		IF (SIf.Cfg.bolEnableLampTest) THEN
			//--------------------------------------------------------------------------------------
			// sub state machine for lamp test sequence
			CASE me.SubStateMachine.intState OF
				cSTA_SUB_INITIALIZED:
					me.SubStateMachine.intStateNext := cSTA_SUB_TestGreen;
				cSTA_SUB_TestGreen:
					SIf.Out.bolGreen.intern := TRUE;
					IF (me.SubStateMachine.udiTimeInState_ms > SIf.Par.udiLampTestTime_ms) THEN 
						me.SubStateMachine.intStateNext := cSTA_SUB_TestYellow;
					END_IF
				cSTA_SUB_TestYellow:
					SIf.Out.bolYellow.intern := TRUE;
					IF (me.SubStateMachine.udiTimeInState_ms > SIf.Par.udiLampTestTime_ms) THEN 
						me.SubStateMachine.intStateNext := cSTA_SUB_TestRed;
					END_IF			
				cSTA_SUB_TestRed:
					SIf.Out.bolRed.intern := TRUE;
					IF (me.SubStateMachine.udiTimeInState_ms > SIf.Par.udiLampTestTime_ms) THEN 
						me.SubStateMachine.intStateNext := cSTA_SUB_TestBeep;
					END_IF				
				cSTA_SUB_TestBeep:
					SIf.Out.bolBeep.intern := TRUE;
					IF (me.SubStateMachine.udiTimeInState_ms > SIf.Par.udiLampTestTime_ms) THEN
						SIf.Out.bolGreen.intern := FALSE;
						SIf.Out.bolYellow.intern := FALSE;
						SIf.Out.bolRed.intern := FALSE;
						SIf.Out.bolBeep.intern := FALSE; 
						me.SubStateMachine.intStateNext := cSTA_SUB_FINISH;
					END_IF				
				cSTA_SUB_FINISH:
					;
				
			END_CASE
		ELSE // Lamp test not enabled, PONBusy is done
			me.SubStateMachine.intStateNext := cSTA_SUB_FINISH;
		END_IF

		
		// State Change Condition
		IF (me.SubStateMachine.intState = cSTA_SUB_FINISH) THEN	// Test done
			me.StateMachine.intStateNext :=  cSTA_PON;
		END_IF
	END_IF




//--------------------------------------------------------------------------------------
// Exit action
	IF (me.StateMachine.intState<>me.StateMachine.intStateNext) THEN
		;
	END_IF
END_METHOD

METHOD PROTECTED sta_RUN : BOOL
// state implemetation
//--------------------------------------------------------------------------------------
// Entry action
	IF (me.StateMachine.intState<>me.StateMachine.intStateLastCycle) THEN
		me.StateMachine.intStateLastCycle := me.StateMachine.intState;

	END_IF


//--------------------------------------------------------------------------------------
// Cyclic action
	IF (me.StateMachine.intState=me.StateMachine.intStateLastCycle) THEN

		// Simulation
		IF (CIf.SwCfg.bolSimulation) THEN
			;
		END_IF
		
		// Oscillator for blinking lamp
		IF (udiTimer >= 2*SIf.Par.udiBlinkTime_ms) THEN
			bolTimer:= FALSE;
			udiTimer:= 0;
		ELSIF (udiTimer >= SIf.Par.udiBlinkTime_ms) THEN
			bolTimer:= TRUE;
		END_IF
		udiTimer:= udiTimer + me.FUBInfo.udiSample_ms;
		// Oscillator for Beep
		IF (udiBeepTimer >= (SIf.Par.udiBeepOffTime_ms + SIf.Par.udiBeepOnTime_ms)) THEN
			bolBeepTimer:= TRUE;
			udiBeepTimer:= 0;
		ELSIF (udiBeepTimer >= SIf.Par.udiBeepOnTime_ms) THEN
			bolBeepTimer:= FALSE;
		END_IF
		udiBeepTimer:= udiBeepTimer + me.FUBInfo.udiSample_ms;	
		
		// Green Lamp
		SIf.Out.bolGreen.intern := setLampOutput(bolBlink:= In_bolGreenBlink, bolOn:= In_bolGreenOn, uinCnt:= In_uinCntGreen, 
												uinCntOLD:= uin_InCntGreenOld, bolOscillator:= bolTimer);
		// Yellow Lamp
		SIf.Out.bolYellow.intern := setLampOutput(bolBlink:= In_bolYellowBlink, bolOn:= In_bolYellowOn, uinCnt:= In_uinCntYellow, 
												uinCntOLD:= uin_InCntYellowOld, bolOscillator:= bolTimer);
		// Red Lamp
		SIf.Out.bolRed.intern := setLampOutput(bolBlink:= In_bolRedBlink, bolOn:= In_bolRedOn, uinCnt:= In_uinCntRed, 
												uinCntOLD:= uin_InCntRedOld, bolOscillator:= bolTimer);
		// Beep										
		SIf.Out.bolBeep.intern := setBeepOutput(bolOscillate:= In_bolBeepOn, uinCnt:= In_uinCntBeep,
												uinCntOLD:= uin_InCntBeepOld, bolOscillator:= bolBeepTimer);
												
		// Reset
		IF (CIf.Job.bolAlmReset) THEN
			uin_InCntGreenOld:= In_uinCntGreen;
			uin_InCntYellowOld:= In_uinCntYellow;
			uin_InCntRedOld:= In_uinCntRed;
			uin_InCntBeepOld:= In_uinCntBeep;
			CIf.Job.bolAlmReset := FALSE;
		END_IF
		
		// State Change Condition
		IF(me.intCmd=cCMD_OFF) THEN
			me.StateMachine.intStateNext := cSTA_OFFBusy;
		END_IF
	END_IF



//--------------------------------------------------------------------------------------
// Exit action
	IF (me.StateMachine.intState<>me.StateMachine.intStateNext) THEN
		;
	END_IF
END_METHOD

METHOD PROTECTED sta_RUNBusy : BOOL
// state implemetation
//--------------------------------------------------------------------------------------
// Entry action
	IF (me.StateMachine.intState<>me.StateMachine.intStateLastCycle) THEN
		me.StateMachine.intStateLastCycle := me.StateMachine.intState;

	END_IF


//--------------------------------------------------------------------------------------
// Cyclic action
	IF (me.StateMachine.intState=me.StateMachine.intStateLastCycle) THEN

		
		// State Change Condition
		IF (TRUE) THEN
			me.StateMachine.intStateNext := cSTA_RUN;
		END_IF
	END_IF


//--------------------------------------------------------------------------------------
// Exit action
	IF (me.StateMachine.intState<>me.StateMachine.intStateNext) THEN
		;
	END_IF
END_METHOD

METHOD PROTECTED StateMachine : BOOL
SUPER^.StateMachine();

// main statemachine of base controller
CASE me.StateMachine.intState OF
	cSTA_RUN:
		THIS^.sta_RUN();
	cSTA_RUNBusy:
		THIS^.sta_RUNBusy();
END_CASE;
END_METHOD

END_FUNCTION_BLOCK

// POUs/Controller/Lvl0/UMC [Universal Motor Controller]/FB_UMC
FUNCTION_BLOCK FB_UMC EXTENDS FB_CtrlBase
VAR_INPUT
	In_uinStatus				: UINT;
	In_intMotorActualSpeed		: INT;
	In_uinMotorSetSpeed			: UINT;
	In_strNetId					: AMSNETID;
	In_uintPort					: WORD;
	In_uinECATState				: UINT;
	In_bolEmoOk					: BOOL;
END_VAR
VAR_OUTPUT
	Out_uinControl      	: UINT;
	Out_uinSpeedSetpoint	: UINT;
END_VAR
VAR
	/// Specific interface struct for public access
	SIf					: T_Ctrl_SIf_UMC;
	In_unStatus			: U_UMC_Lenze_Status;
	Out_unControl		: U_UMC_Lenze_Control;
	arTurnDirection		: ARRAY[0..MAX_E_TURN_DIRECTION] OF BOOL;
	fbPulse				: TC2_STANDARD.TP;
END_VAR
VAR CONSTANT
	cLEFT				: BOOL := TRUE;
	cRIGHT				: BOOL := FALSE;

	cEtherCAT_OP_MODE		: UINT := 16#0008;
	cEtherCAT_MODE_MASK		: UINT := 16#000F;
END_VAR

(*__________________________________________________________________________________________________
¦	
¦	Vistaprint Schweiz GmbH
¦	CH - 8401 Winterthur
¦
¦	www.vistaprint.ch - info@vistaprint.ch
¦___________________________________________________________________________________________________

Function desription:
Lenze Motor implementation. 


History:
Version		Date			Author		Comment
---------------------------------------------------------------------------------------------------
0.00.1		09.07.2013		PC			Start history
0.00.2		04.02.2014		AVM/MRU		Simulation mode
										cCMD_LEFT / cCMD_RIGHT added in FB_init / getCmdState

___________________________________________________________________________________________________*)


IF (me.bolActivate) THEN // cyclic call enabled
	IF (CIf.Info.bolInitDone=FALSE) THEN // first cycle -> init
		CtrlInit();
		CIf.Info.bolInitDone := TRUE;
	ELSE
		CycleStartDuty();
	
		Always();
		
		StateMachine();
		
		CycleEndDuty();
	END_IF
END_IF;

METHOD PROTECTED Always : BOOL
SUPER^.Always();

// ----------------------------------------------------------------------------------
// Simulation
IF (CIf.SwCfg.bolSimulation) THEN
	// Simulate inputs (no physical inputs)
	SIf.In.bolEmoOk.intern := TRUE;
END_IF

// ----------------------------------------------------------------------------------
// Conditions Always
IF (me.StateMachine.intState<>cSTA_SINGLE_ANSWER) THEN
	IF (((me.Alarm.eActivAlmClass=E_AlmClass.OFF) OR (me.intCmd=cCMD_OFF))
			AND (me.StateMachine.intState<>cSTA_ERROR) AND (me.StateMachine.intState<>cSTA_ERRORQuit)
			AND (me.StateMachine.intState<>cSTA_EOFF) AND (me.StateMachine.intState<>cSTA_EOFFBusy)
			AND (me.StateMachine.intState<>cSTA_OFF) AND (me.StateMachine.intState<>cSTA_OFFBusy)
			AND (me.StateMachine.intState<>UMC_CmdState.cSTA_RESETMOTORERROR) 
			AND (me.StateMachine.intState<>UMC_CmdState.cSTA_SETOPERATIONMODE)) THEN
		me.StateMachine.intStateNext := cSTA_OFFBusy;	
	END_IF

	//-------------------------------------------------------------------------------
	// Monitoring of inputs from Safety PLC (no physical inputs)
	//-------------------------------------------------------------------------------
	// Emergency Off
	IF ((SIf.In.bolEmoOk.intern = FALSE) AND (me.StateMachine.intState <> cSTA_EOFF) 
		AND (me.StateMachine.intState <> BASE_PLC.cSTA_EOFFBusy)
		AND (me.StateMachine.intState <> BASE_PLC.cSTA_ERROR) 
		AND (me.StateMachine.intState <> BASE_PLC.cSTA_PON) 
		AND (me.StateMachine.intState <> BASE_PLC.cSTA_PONBusy) 
		AND (me.StateMachine.intState<>BASE_PLC.cSTA_INITIALIZED)
		AND (me.StateMachine.intState <> BASE_PLC.cSTA_ERRORQuit)) THEN
		me.StateMachine.intStateNext := cSTA_EOFFBusy;				
	END_IF	
END_IF
END_METHOD

METHOD PROTECTED cmd_MotorOff : BOOL
Out_unControl.Output 				:= 0;
Out_unControl.Data.SetDCBreak 		:= 1;
Out_unControl.Data.SetHalt        	:= 1;
Out_unControl.Data.SetQuickStop    	:= 1;
SIf.Out.uinSpeedSetpoint.intern 	:= 0;
END_METHOD

METHOD PROTECTED cmd_MotorOn : BOOL
VAR_INPUT
	bDirection		: BOOL;		// Direction of the drive; False = Right; True = Left
	uinSpeed		: UINT;					// Speed of the belt
END_VAR
Out_unControl.Output 				:= 0;
Out_unControl.Data.EnableOperation 	:= 1;
Out_unControl.Data.SwitchOn        	:= 1;
Out_unControl.Data.SetSpeedCcw     	:= bDirection;

SIf.Out.uinSpeedSetpoint.intern 	:= uinSpeed;
END_METHOD

METHOD PROTECTED cmd_MotorReset : BOOL
VAR_INPUT
END_VAR
cmd_MotorOff();
Out_unControl.Data.ResetFault 		:= 1;
END_METHOD

METHOD PROTECTED cmd_MotorStop : BOOL
VAR_INPUT
END_VAR
Out_unControl.Output 				:= 0;
Out_unControl.Data.SetDCBreak 		:= 1;
Out_unControl.Data.SetHalt        	:= 1;
Out_unControl.Data.SetQuickStop    	:= 1;
END_METHOD

METHOD PROTECTED CtrlInit : BOOL
VAR_INPUT
END_VAR
SUPER^.CtrlInit();

arTurnDirection[E_TURN_DIRECTION.AUTOMATIC] := FALSE;
arTurnDirection[E_TURN_DIRECTION.LEFT] 		:= FALSE;
arTurnDirection[E_TURN_DIRECTION.RIGHT] 	:= TRUE;

SIf.Cur.uinSpeedLimit := SIf.Cfg.uinMaxSpeed * SIf.Cfg.uinLC11_100 / 100;
END_METHOD

PROPERTY PUBLIC CtrlSIf : POINTER TO T_Ctrl_SIf_UMC
GET
CtrlSIf := ADR(SIf);
END_GET
SET
END_SET
END_PROPERTY

METHOD PROTECTED CycleEndDuty : BOOL
VAR_INPUT
END_VAR
SIf.Out.uinControl.intern := Out_unControl.Output;

SUPER^.CycleEndDuty();
END_METHOD

METHOD PROTECTED CycleStartDuty : BOOL
VAR_INPUT
END_VAR
SUPER^.CycleStartDuty();

In_unStatus.Input := SIf.In.uinStatus.intern;
END_METHOD

METHOD FB_init : BOOL
VAR_INPUT
	bInitRetains : BOOL; // if TRUE, the retain variables are initialized (warm start / cold start)
	bInCopyCode : BOOL;  // if TRUE, the instance afterwards gets moved into the copy code (online change)
END_VAR
VAR
	iIdx		: UINT;
	iLength		: UINT;	
END_VAR
//------------------------------------------------------------------------------------------------------------------------
// to manually change in new FUB implementation!!!
// define valid commands for this controller
iLength := SIZEOF(CIf.Job.aCmdList)/SIZEOF(CIf.Job.aCmdList[0]);
iIdx := 0;

WHILE (iIdx < iLength) AND (CIf.Job.aCmdList[iIdx].intCmd <> cCMD_INITIALIZED) DO
	iIdx := iIdx + 1; 
END_WHILE

IF (iIdx < iLength) THEN
// Add configuration of own comands	
	CIf.Job.aCmdList[iIdx].intCmd := BASE_PLC.cCMD_STOP;
	CIf.Job.aCmdList[iIdx].strName := 'Stop'; 
	CIf.Job.aCmdList[iIdx].bolAvailable := TRUE;
	iIdx := iIdx + 1;
	CIf.Job.aCmdList[iIdx].intCmd := cCMD_RUN;
	CIf.Job.aCmdList[iIdx].strName := 'Run'; 
	CIf.Job.aCmdList[iIdx].bolAvailable := TRUE;
	iIdx := iIdx + 1;
	CIf.Job.aCmdList[iIdx].intCmd := cCMD_LEFT;
	CIf.Job.aCmdList[iIdx].strName := 'Left'; 
	CIf.Job.aCmdList[iIdx].bolAvailable := TRUE;
	iIdx := iIdx + 1;
	CIf.Job.aCmdList[iIdx].intCmd := cCMD_RIGHT;
	CIf.Job.aCmdList[iIdx].strName := 'Right'; 
	CIf.Job.aCmdList[iIdx].bolAvailable := TRUE;
	iIdx := iIdx + 1;
ELSE
	;// Error if the aCmdList Array is to small
END_IF

// set name of class/typ
CIf.Info.strType := 'FB_UMC'; 

// set alarm class
SIf.Alm[E_ALM_UMC.MotorOnTimeout].eAlmClass := Base_PLC.E_AlmClass.TSTOP;
SIf.Alm[E_ALM_UMC.MotorOnTimeout].strText := 'Motor On Timeout'; 
SIf.Alm[E_ALM_UMC.MotorError].eAlmClass := Base_PLC.E_AlmClass.TSTOP;
SIf.Alm[E_ALM_UMC.MotorError].strText := 'Motor Error';
SIf.Alm[E_ALM_UMC.MotorWarning].eAlmClass := Base_PLC.E_AlmClass.WARNING;
SIf.Alm[E_ALM_UMC.MotorWarning].strText := 'Motor Warning';
SIf.Alm[E_ALM_UMC.MotorOverCurrent].eAlmClass := Base_PLC.E_AlmClass.WARNING;
SIf.Alm[E_ALM_UMC.MotorOverCurrent].strText := 'Motor Over Current';
SIf.Alm[E_ALM_UMC.MotorNotReady].eAlmClass := Base_PLC.E_AlmClass.TSTOP;
SIf.Alm[E_ALM_UMC.MotorNotReady].strText := 'Motor Not Ready';
SIf.Alm[E_ALM_UMC.DirectionParameterOverflow].eAlmClass := Base_PLC.E_AlmClass.TSTOP;
SIf.Alm[E_ALM_UMC.DirectionParameterOverflow].strText := 'Direction Parameter Overflow';
SIf.Alm[E_ALM_UMC.SpeedOverLimit].eAlmClass := Base_PLC.E_AlmClass.WARNING;
SIf.Alm[E_ALM_UMC.SpeedOverLimit].strText := 'Motor Setpoint over the limit';

//*******************************************************************************
// initial values
//*******************************************************************************

// software configuration
CIf.SwCfg.bolExist := TRUE;
CIf.SwCfg.bolEnable := TRUE;
CIf.SwCfg.bolSimulation := FALSE;

// configuration
SIf.Cfg.uinLC11 := 1500;
SIf.Cfg.uinLC11_100 := 16384;
SIf.Cfg.uinMaxSpeed := 150;

// parameter
SIf.Par.udiStartupOnTime_ms := 5000;
SIf.Par.udiMotorOnTime_ms 	:= 10000;
SIf.Par.uinSpeed_rpm 		:= 1000;
SIf.Par.uinMotorResetPulseTime_ms	:= 500;
SIf.Par.uinMotorResetCnt 		:= 3;
SIf.Par.udiMoveStartLatency 	:= 15;
SIf.Par.udiMoveStopLatency 		:= 60;
SIf.Par.eRotationDirection  := E_TURN_DIRECTION.LEFT;

SIf.Par.udiSimMotorOnTime_ms := SIf.Par.udiMotorOnTime_ms / 10;
END_METHOD

METHOD PROTECTED getCmdState : STRING

VAR_INPUT
	intCmdState: INT;
	bolState: BOOL;
END_VAR
getCmdState := SUPER^.getCmdState(intCmdState:=intCmdState,bolState:=bolState); // get global/base defined cmds/states

IF (getCmdState='') THEN // global not defined get local
	// get string cmd/state string information in runtime
	IF (bolState=FALSE) THEN
		// Comands's
		CASE intCmdState OF
			cCMD_LEFT: 
				getCmdState := 'cCMD_Left';
			cCMD_RIGHT: 
				getCmdState := 'cCMD_Right';
		END_CASE;
	ELSE
		// States's
		CASE intCmdState OF
			cSTA_RUN: 
				getCmdState := 'RUN';
			cSTA_RUNBusy: 
				getCmdState := 'RUNBusy';
			UMC_CmdState.cSTA_RESETMOTORERROR:
				getCmdState := 'RESETMOTORERROR';
			UMC_CmdState.cSTA_SETOPERATIONMODE:
				getCmdState := 'SETOPERATIONMODE';
		END_CASE;
	END_IF
END_IF
END_METHOD

METHOD getCtrlSIf : POINTER TO T_Ctrl_SIf_UMC
getCtrlSIf := ADR(SIf);
END_METHOD

METHOD PROTECTED GetMotorStatus : E_UMC_MOTOR_STATUS
VAR_INPUT
	uinMotorStatus		: UINT;
END_VAR
uinMotorStatus := uinMotorStatus AND 16#0F00;
uinMotorStatus := SHR(uinMotorStatus,8);
GetMotorStatus := UINT_TO_INT(uinMotorStatus);
END_METHOD

METHOD PROTECTED GetSpeedValue : UINT
VAR
	uinSpeedOutput			: UINT;
END_VAR
uinSpeedOutput := SIf.Par.uinSpeed_rpm * SIf.Cfg.uinLC11_100 / SIf.Cfg.uinLC11;

IF uinSpeedOutput > SIf.Cur.uinSpeedLimit THEN
	uinSpeedOutput := SIf.Cur.uinSpeedLimit;
	pfbAlarmCtrl^.setAlarm(CIf.Info.intCtrlId,INT_TO_UINT(E_ALM_UMC.SpeedOverLimit),0,ADR(SIf.Alm),E_AlmState.RST,CIf.Job.eMe_ActivAlmClass);
END_IF

GetSpeedValue := uinSpeedOutput;
END_METHOD

METHOD PROTECTED IoInBridge : BOOL
// digitale and analoge inputs read from hardware or forcing
SIf.In.uinStatus.map			:= THIS^.In_uinStatus				;
SIf.In.intMotorActualSpeed.map	:= THIS^.In_intMotorActualSpeed	;
SIf.In.uinMotorSetSpeed.map		:= THIS^.In_uinMotorSetSpeed		;
SIf.In.bolEmoOk.map				:= THIS^.In_bolEmoOk		;

IF (CIf.SwCfg.bolSimulation = FALSE) THEN
	BASE_PLC.getInUint(CIf.Job.bolIoForce,ADR(SIf.In.uinStatus));
	BASE_PLC.getInUint(CIf.Job.bolIoForce,ADR(SIf.In.intMotorActualSpeed));
	BASE_PLC.getInUint(CIf.Job.bolIoForce,ADR(SIf.In.uinMotorSetSpeed));
	BASE_PLC.getInUint(CIf.Job.bolIoForce,ADR(SIf.In.bolEmoOk));
ELSE
	//simulation of global IO
END_IF
END_METHOD

METHOD PROTECTED IoOutBridge : BOOL
VAR
	bolSwitchValvesOff: BOOL;
END_VAR
// digitale and analoge inputs read from hardware or forcing
IF (CIf.SwCfg.bolSimulation = FALSE) THEN
	BASE_PLC.setOutUint(CIf.Job.bolIoForce ,ADR(SIf.Out.uinControl));
	BASE_PLC.setOutUint(CIf.Job.bolIoForce ,ADR(SIf.Out.uinSpeedSetpoint));

	THIS^.Out_uinControl			:= SIf.Out.uinControl.map	;
	THIS^.Out_uinSpeedSetpoint		:= SIf.Out.uinSpeedSetpoint.map	;
END_IF
END_METHOD

METHOD PROTECTED sta_EOFF : BOOL
VAR_INPUT
END_VAR
// state implemetation
//--------------------------------------------------------------------------------------
// Entry action
	IF (me.StateMachine.intState<>me.StateMachine.intStateLastCycle) THEN
		me.StateMachine.intStateLastCycle := me.StateMachine.intState;	
	END_IF

//--------------------------------------------------------------------------------------
// Cyclic action
	IF (me.StateMachine.intState=me.StateMachine.intStateLastCycle) THEN		
		// As long as the EMO is not reseted!
		IF SIf.In.bolEmoOk.intern THEN
			me.StateMachine.intStateNext := BASE_PLC.cSTA_OFFBusy;			
		ELSE
			IF me.intCmd <> BASE_PLC.cCMD_OFF THEN
				// Clear pending and new commands cyclic to prevent automatic recovery!	
				CIf.Job.intACmd := BASE_PLC.cCMD_DONE;
				CIf.Job.intMCmd := BASE_PLC.cCMD_DONE;		
			END_IF
		END_IF
	END_IF

//--------------------------------------------------------------------------------------
// Exit action
	IF (me.StateMachine.intState<>me.StateMachine.intStateNext) THEN
		;
	END_IF
END_METHOD

METHOD PROTECTED sta_EOFFbusy : BOOL
VAR_INPUT
END_VAR
// state implemetation
//--------------------------------------------------------------------------------------
// Entry action
IF (me.StateMachine.intState<>me.StateMachine.intStateLastCycle) THEN
	me.StateMachine.intStateLastCycle := me.StateMachine.intState;
	cmd_MotorOff();
END_IF

//--------------------------------------------------------------------------------------
// Cyclic action
IF (me.StateMachine.intState=me.StateMachine.intStateLastCycle) THEN
	IF (TRUE) THEN
		me.StateMachine.intStateNext := BASE_PLC.cSTA_EOFF;
	END_IF
END_IF

//--------------------------------------------------------------------------------------
// Exit action
IF (me.StateMachine.intState<>me.StateMachine.intStateNext) THEN
	;
END_IF
END_METHOD

METHOD PROTECTED sta_ERROR : BOOL
// state implemetation
//--------------------------------------------------------------------------------------
// Entry action
	IF (me.StateMachine.intState<>me.StateMachine.intStateLastCycle) THEN
		me.StateMachine.intStateHistory := me.StateMachine.intStateLastCycle; // -> possibillity to go back to state before error
		me.StateMachine.intStateLastCycle := me.StateMachine.intState;
		SIf.Cur.uinMotorResetCnt := 0;
		cmd_MotorOff();
	END_IF


//--------------------------------------------------------------------------------------
// Cyclic action
	IF (me.StateMachine.intState=me.StateMachine.intStateLastCycle) THEN
		
		;
		
		
		// State Change Condition
		IF (CIf.Job.bolAlmReset = TRUE) THEN
			me.StateMachine.intStateNext := cSTA_ERRORQuit;
		END_IF
	END_IF




//--------------------------------------------------------------------------------------
// Exit action
	IF (me.StateMachine.intState<>me.StateMachine.intStateNext) THEN
		;
	END_IF
END_METHOD

METHOD PROTECTED sta_ERRORQuit : BOOL
// state implemetation
//--------------------------------------------------------------------------------------
// Entry action
	IF (me.StateMachine.intState<>me.StateMachine.intStateLastCycle) THEN
		me.StateMachine.intStateLastCycle := me.StateMachine.intState;
		
	END_IF


//--------------------------------------------------------------------------------------
// Cyclic action
	IF (me.StateMachine.intState=me.StateMachine.intStateLastCycle) THEN
		
		;
		// evtl. wait time if reset of device is necessary and then decide to go to states or ERROR state
		IF (CIf.Job.bolAlmReset = TRUE) THEN
			CIf.Job.eMe_ActivAlmClass := E_AlmClass.NONE; // reset feedback channel for parent
			CIf.Job.bolAlmReset := FALSE;
		END_IF
		
		// State Change Condition
		IF (CIf.Job.bolAlmReset = FALSE) THEN
			IF (me.StateMachine.intStateHistory<=cSTA_PON) THEN
				me.StateMachine.intStateNext := cSTA_PON;
			ELSIF (CIf.SwCfg.bolSimulation = TRUE) THEN	// Do not set operation mode in simulation
				me.StateMachine.intStateNext := BASE_PLC.cSTA_OFF;
			ELSE
				me.StateMachine.intStateNext := UMC_CmdState.cSTA_SETOPERATIONMODE;
			END_IF
		END_IF
	END_IF




//--------------------------------------------------------------------------------------
// Exit action
	IF (me.StateMachine.intState<>me.StateMachine.intStateNext) THEN
		;
	END_IF
END_METHOD

METHOD PROTECTED sta_OFF : BOOL
VAR_INPUT
END_VAR
// state implemetation
//--------------------------------------------------------------------------------------
// Entry action
	IF (me.StateMachine.intState<>me.StateMachine.intStateLastCycle) THEN
		me.StateMachine.intStateLastCycle := me.StateMachine.intState;

		SIf.Cur.uinMotorResetCnt := 0;
	END_IF


//--------------------------------------------------------------------------------------
// Cyclic action
	IF (me.StateMachine.intState=me.StateMachine.intStateLastCycle) THEN
		CASE me.intCmd OF
			cCMD_Left:
				SIf.Par.eRotationDirection := E_TURN_DIRECTION.LEFT;
				me.StateMachine.intStateNext := cSTA_RUNBusy;
			cCMD_Right:
				SIf.Par.eRotationDirection := E_TURN_DIRECTION.RIGHT;
				me.StateMachine.intStateNext := cSTA_RUNBusy;
			BASE_PLC.cCMD_STOP:
				me.StateMachine.intStateNext := BASE_PLC.cSTA_STOPBusy;
			BASE_PLC.cCMD_RUN:
				me.StateMachine.intStateNext := cSTA_RUNBusy;
		END_CASE
	END_IF


//--------------------------------------------------------------------------------------
// Exit action
	IF (me.StateMachine.intState<>me.StateMachine.intStateNext) THEN
		;
	END_IF
END_METHOD

METHOD PROTECTED sta_OFFBusy : BOOL
VAR
	uinECatStatus	: UINT;
	eMotorStatus	: E_UMC_MOTOR_STATUS;
END_VAR
// state implemetation
//--------------------------------------------------------------------------------------
// Entry action
	IF (me.StateMachine.intState<>me.StateMachine.intStateLastCycle) THEN
		me.StateMachine.intStateLastCycle := me.StateMachine.intState;
		cmd_MotorOff();
	END_IF


//--------------------------------------------------------------------------------------
// Cyclic action
	IF (me.StateMachine.intState=me.StateMachine.intStateLastCycle) THEN
		eMotorStatus := GetMotorStatus(sif.In.uinStatus.intern);
		uinECatStatus := In_uinECATState AND cEtherCAT_MODE_MASK;

		IF    (uinECatStatus = cEtherCAT_OP_MODE)
		  AND NOT In_unStatus.Data.Trouble 
		  AND In_unStatus.Data.ActSpeedIsZero
		  AND (eMotorStatus = E_UMC_MOTOR_STATUS.ReadyToSwitchON) THEN
			me.StateMachine.intStateNext := Base_PLC.cSTA_OFF;
		ELSIF (CIf.SwCfg.bolSimulation = TRUE) THEN	// Do not set operation mode in simulation
			me.StateMachine.intStateNext := BASE_PLC.cSTA_OFF;
		ELSE
			IF me.StateMachine.udiTimeInState_ms > SIf.Par.uinMotorResetPulseTime_ms THEN
				IF SIf.Cur.uinMotorResetCnt > SIf.Par.uinMotorResetCnt THEN
					pfbAlarmCtrl^.setAlarm(CIf.Info.intCtrlId,INT_TO_UINT(E_ALM_UMC.MotorError),0,ADR(SIf.Alm),E_AlmState.RST,CIf.Job.eMe_ActivAlmClass);
					me.StateMachine.intStateNext := Base_PLC.cSTA_ERROR;	
				ELSE
					me.StateMachine.intStateNext := UMC_CmdState.cSTA_SETOPERATIONMODE;
				END_IF
			END_IF
		END_IF
	END_IF

//--------------------------------------------------------------------------------------
// Exit action
	IF (me.StateMachine.intState<>me.StateMachine.intStateNext) THEN
		;
	END_IF
END_METHOD

METHOD PROTECTED sta_PON : BOOL
VAR_INPUT
END_VAR
// state implemetation
//--------------------------------------------------------------------------------------
// Entry action
	IF (me.StateMachine.intState<>me.StateMachine.intStateLastCycle) THEN
		me.StateMachine.intStateLastCycle := me.StateMachine.intState;
		
	END_IF


//--------------------------------------------------------------------------------------
// Cyclic action
	IF (me.StateMachine.intState=me.StateMachine.intStateLastCycle) THEN
		;
	END_IF




//--------------------------------------------------------------------------------------
// Exit action
	IF (me.StateMachine.intState<>me.StateMachine.intStateNext) THEN
		;
	END_IF
END_METHOD

METHOD PROTECTED sta_RESETMOTORERROR : BOOL
VAR
	eMotorStatus	: E_UMC_MOTOR_STATUS;
END_VAR
// state implemetation
//--------------------------------------------------------------------------------------
// Entry action
	IF (me.StateMachine.intState<>me.StateMachine.intStateLastCycle) THEN
		me.StateMachine.intStateLastCycle := me.StateMachine.intState;
		cmd_MotorReset();
	END_IF


//--------------------------------------------------------------------------------------
// Cyclic action
	IF (me.StateMachine.intState=me.StateMachine.intStateLastCycle) THEN
		eMotorStatus := GetMotorStatus(sif.In.uinStatus.intern);

		IF me.SubStateMachine.udiTimeInState_ms > SIf.Par.uinMotorResetPulseTime_ms THEN
			SIf.Cur.uinMotorResetCnt := SIf.Cur.uinMotorResetCnt + 1;
			me.StateMachine.intStateNext := BASE_PLC.cSTA_OFFBusy;
		END_IF
	END_IF


//--------------------------------------------------------------------------------------
// Exit action
	IF (me.StateMachine.intState<>me.StateMachine.intStateNext) THEN
		Out_unControl.Data.ResetFault := FALSE;
	END_IF
END_METHOD

METHOD PROTECTED sta_RUN : BOOL
VAR
	uniStatus 		: U_UMC_Lenze_Status;
END_VAR
// state implemetation
//--------------------------------------------------------------------------------------
// Entry action
	IF (me.StateMachine.intState<>me.StateMachine.intStateLastCycle) THEN
		me.StateMachine.intStateLastCycle := me.StateMachine.intState;
		CIf.Job.intACmd := BASE_PLC.cCMD_DONE;
	END_IF


//--------------------------------------------------------------------------------------
// Cyclic action
	IF (me.StateMachine.intState=me.StateMachine.intStateLastCycle) THEN
		IF In_unStatus.Data.Trouble THEN
			pfbAlarmCtrl^.setAlarm(CIf.Info.intCtrlId,INT_TO_UINT(E_ALM_UMC.MotorError),0,ADR(SIf.Alm),E_AlmState.RST,CIf.Job.eMe_ActivAlmClass);
			me.StateMachine.intStateNext := Base_PLC.cSTA_ERROR;	
		END_IF
		
		IF (me.StateMachine.intStateNext <> Base_PLC.cSTA_ERROR) THEN
			// Reenter the RunBusy state again if the speed changes
			IF SIf.Par.uinSpeed_rpm <> SIf.Cur.uinSpeed_rpm THEN
				me.StateMachine.intStateNext := cSTA_RUNBusy;
			END_IF
			
			// Reenter the RunBusy state again if the direction changes.
			IF SIf.Par.eRotationDirection <> SIf.Cur.eDirection THEN
				me.StateMachine.intStateNext := cSTA_RUNBusy;
			END_IF

			CASE me.intCmd OF
				cCMD_Left:
					SIf.Par.eRotationDirection := E_TURN_DIRECTION.LEFT;
					me.StateMachine.intStateNext := cSTA_RUNBusy;
				cCMD_Right:
					SIf.Par.eRotationDirection := E_TURN_DIRECTION.RIGHT;
					me.StateMachine.intStateNext := cSTA_RUNBusy;
				BASE_PLC.cCMD_STOP:
					me.StateMachine.intStateNext := BASE_PLC.cSTA_STOPBusy;
			END_CASE
		END_IF
END_IF


//--------------------------------------------------------------------------------------
// Exit action
	IF (me.StateMachine.intState<>me.StateMachine.intStateNext) THEN
		;
	END_IF
END_METHOD

METHOD PROTECTED sta_RUNBusy : BOOL
VAR
	uniStatus 		: U_UMC_Lenze_Status;
END_VAR
// state implemetation
//--------------------------------------------------------------------------------------
// Entry action
	IF (me.StateMachine.intState<>me.StateMachine.intStateLastCycle) THEN
		me.StateMachine.intStateLastCycle := me.StateMachine.intState;

		SIf.Cur.uinSpeed_rpm := SIf.Par.uinSpeed_rpm;
		SIf.Cur.uinSpeedOuput := GetSpeedValue();
		SIf.Cur.eDirection 	:= SIf.Par.eRotationDirection;
		
		// Switch Motor ON
		IF SIf.Par.eRotationDirection < E_TURN_DIRECTION.MAX_E_TURN_DIRECTION THEN
			cmd_MotorOn(arTurnDirection[SIf.Par.eRotationDirection], SIf.Cur.uinSpeedOuput);
		ELSE
			pfbAlarmCtrl^.setAlarm(CIf.Info.intCtrlId,INT_TO_UINT(E_ALM_UMC.DirectionParameterOverflow),0,ADR(SIf.Alm),E_AlmState.RST,CIf.Job.eMe_ActivAlmClass);
			me.StateMachine.intStateNext := Base_PLC.cSTA_ERROR;	
		END_IF

		fbSimulationTimer.IN := FALSE;
		fbSimulationTimer.PT := UDINT_TO_TIME(SIf.Par.udiSimMotorOnTime_ms);
		fbSimulationTimer(); // set time/reset timer
		fbSimulationTimer.IN := TRUE; // start timer

	END_IF


//--------------------------------------------------------------------------------------
// Cyclic action
	IF (me.StateMachine.intState=me.StateMachine.intStateLastCycle) THEN
		IF (CIf.SwCfg.bolSimulation) THEN
			fbSimulationTimer(); // simulation time
			IF (fbSimulationTimer.Q) THEN
				SIf.In.uinMotorSetSpeed.intern 	:= SIf.Out.uinSpeedSetpoint.intern;
				SIf.In.uinMotorSetSpeed.intern 	:= SIf.Out.uinSpeedSetpoint.intern;
				uniStatus.Input 				:= 0;
				uniStatus.Data.DriveReady		:= 1;
				uniStatus.Data.SpeedActEqualSet := 1;
				uniStatus.Data.SpeedSetReached  := 1;
				uniStatus.Data.Status_1			:= 1;
				uniStatus.Data.Status_3			:= 1;
				uniStatus.Data.SpeedCcw			:= arTurnDirection[SIf.Par.eRotationDirection];
				SIf.In.uinStatus.intern 		:= uniStatus.Input;
			END_IF
		END_IF

		IF (me.StateMachine.udiTimeInState_ms > SIf.Par.udiMotorOnTime_ms) THEN
			pfbAlarmCtrl^.setAlarm(CIf.Info.intCtrlId,INT_TO_UINT(E_ALM_UMC.MotorOnTimeout),0,ADR(SIf.Alm),E_AlmState.RST,CIf.Job.eMe_ActivAlmClass);
			me.StateMachine.intStateNext := Base_PLC.cSTA_ERROR;	
		END_IF

		IF In_unStatus.Data.Trouble THEN
			pfbAlarmCtrl^.setAlarm(CIf.Info.intCtrlId,INT_TO_UINT(E_ALM_UMC.MotorError),0,ADR(SIf.Alm),E_AlmState.RST,CIf.Job.eMe_ActivAlmClass);
			me.StateMachine.intStateNext := Base_PLC.cSTA_ERROR;	
		END_IF
		
		IF (me.StateMachine.intStateNext <> Base_PLC.cSTA_ERROR) THEN
			IF (NOT In_unStatus.Data.Trouble) 
				AND (THIS^.arTurnDirection[SIf.Cur.eDirection] = In_unStatus.Data.SpeedCcw)	THEN
//				AND (In_unStatus.Data.SpeedSetReached) THEN
				me.StateMachine.intStateNext := cSTA_RUN;
			END_IF;	

			// Reenter the RunBusy state again if the speed changes
			IF GetSpeedValue() <> SIf.Cur.uinSpeedOuput THEN
				me.StateMachine.intStateLastCycle := -1;
			END_IF
			
			// Reenter the RunBusy state again if the direction changes.
			IF SIf.Par.eRotationDirection <> SIf.Cur.eDirection THEN
				me.StateMachine.intStateLastCycle := -1;
			END_IF
			
			CASE me.intCmd OF
				cCMD_Left:
					IF SIf.Par.eRotationDirection <> E_TURN_DIRECTION.LEFT THEN
						SIf.Par.eRotationDirection := E_TURN_DIRECTION.LEFT;
						me.StateMachine.intStateLastCycle := -1;
					END_IF
				cCMD_Right:
					IF SIf.Par.eRotationDirection <> E_TURN_DIRECTION.RIGHT THEN
						SIf.Par.eRotationDirection := E_TURN_DIRECTION.RIGHT;
						me.StateMachine.intStateLastCycle := -1;
					END_IF
				BASE_PLC.cCMD_STOP:
					me.StateMachine.intStateNext := BASE_PLC.cSTA_STOPBusy;
			END_CASE
		END_IF
END_IF


//--------------------------------------------------------------------------------------
// Exit action
	IF (me.StateMachine.intState<>me.StateMachine.intStateNext) THEN
		;
	END_IF
END_METHOD

METHOD PROTECTED sta_SETOPERATIONMODE : BOOL
VAR
	uinECatStatus		: UINT;

	fbEcReqSlaveState 	: FB_EcReqSlaveState;
	bExecute        	: BOOL;
	uinReqState     	: WORD := EC_DEVICE_STATE_OP;
	bError          	: BOOL;
	nErrId          	: UDINT;
END_VAR
// state implemetation
//--------------------------------------------------------------------------------------
// Entry action
	IF (me.StateMachine.intState<>me.StateMachine.intStateLastCycle) THEN
		me.StateMachine.intStateLastCycle := me.StateMachine.intState;
	END_IF


//--------------------------------------------------------------------------------------
// Cyclic action
	IF (me.StateMachine.intState=me.StateMachine.intStateLastCycle) THEN
		bExecute := NOT ((In_uinECATState AND cEtherCAT_MODE_MASK) = cEtherCAT_OP_MODE);

		IF NOT bExecute THEN
			me.StateMachine.intStateNext := UMC_CmdState.cSTA_RESETMOTORERROR;
		END_IF

		fbEcReqSlaveState(
			sNetId		:= F_CreateAmsNetId(In_strNetId), 
			nSlaveAddr	:= In_uintPort, 
			bExecute	:= bExecute, 
			state		:= uinReqState  );

		IF (me.StateMachine.udiTimeInState_ms > SIf.Par.udiStartupOnTime_ms) THEN
			pfbAlarmCtrl^.setAlarm(CIf.Info.intCtrlId,INT_TO_UINT(E_ALM_UMC.MotorError),0,ADR(SIf.Alm),E_AlmState.RST,CIf.Job.eMe_ActivAlmClass);
			me.StateMachine.intStateNext := Base_PLC.cSTA_ERROR;	
		END_IF
END_IF


//--------------------------------------------------------------------------------------
// Exit action
	IF (me.StateMachine.intState<>me.StateMachine.intStateNext) THEN
		Out_unControl.Data.ResetFault := FALSE;
	END_IF
END_METHOD

METHOD PROTECTED sta_STOP : BOOL
VAR_INPUT
END_VAR
// state implemetation
//--------------------------------------------------------------------------------------
// Entry action
	IF (me.StateMachine.intState<>me.StateMachine.intStateLastCycle) THEN
		me.StateMachine.intStateLastCycle := me.StateMachine.intState;

	END_IF


//--------------------------------------------------------------------------------------
// Cyclic action
	IF (me.StateMachine.intState=me.StateMachine.intStateLastCycle) THEN
		CASE me.intCmd OF
			cCMD_Left:
				SIf.Par.eRotationDirection := E_TURN_DIRECTION.LEFT;
				me.StateMachine.intStateNext := cSTA_RUNBusy;
			cCMD_Right:
				SIf.Par.eRotationDirection := E_TURN_DIRECTION.RIGHT;
				me.StateMachine.intStateNext := cSTA_RUNBusy;
			BASE_PLC.cCMD_RUN:
				me.StateMachine.intStateNext := cSTA_RUNBusy;
		END_CASE
	END_IF


//--------------------------------------------------------------------------------------
// Exit action
	IF (me.StateMachine.intState<>me.StateMachine.intStateNext) THEN
		;
	END_IF
END_METHOD

METHOD PROTECTED sta_STOPBusy : BOOL
VAR
	uniStatus 		: U_UMC_Lenze_Status;
END_VAR
// state implemetation
//--------------------------------------------------------------------------------------
// Entry action
	IF (me.StateMachine.intState<>me.StateMachine.intStateLastCycle) THEN
		me.StateMachine.intStateLastCycle := me.StateMachine.intState;
		// Switch Motor Off
		cmd_MotorStop();
	END_IF


//--------------------------------------------------------------------------------------
// Cyclic action
	IF (me.StateMachine.intState=me.StateMachine.intStateLastCycle) THEN
		IF (CIf.SwCfg.bolSimulation) THEN
			SIf.In.uinMotorSetSpeed.intern 	:= 0;
			SIf.In.intMotorActualSpeed.intern 	:= 0;
			uniStatus.Input 				:= 0;
			uniStatus.Data.ActSpeedIsZero	:= TRUE;
			SIf.In.uinStatus.intern 		:= uniStatus.Input;
		END_IF

		IF (me.StateMachine.udiTimeInState_ms < SIf.Par.udiMotorOnTime_ms) THEN
			IF (NOT In_unStatus.Data.Trouble) AND (In_unStatus.Data.ActSpeedIsZero) THEN
				me.StateMachine.intStateNext := Base_PLC.cSTA_STOP;
			END_IF;	
		ELSE
			pfbAlarmCtrl^.setAlarm(CIf.Info.intCtrlId,INT_TO_UINT(E_ALM_UMC.MotorError),0,ADR(SIf.Alm),E_AlmState.RST,CIf.Job.eMe_ActivAlmClass);
			me.StateMachine.intStateNext := Base_PLC.cSTA_ERROR;	
		END_IF
END_IF


//--------------------------------------------------------------------------------------
// Exit action
	IF (me.StateMachine.intState<>me.StateMachine.intStateNext) THEN
		Out_unControl.Data.ResetFault := FALSE;
	END_IF
END_METHOD

METHOD PROTECTED StateMachine : BOOL
SUPER^.StateMachine();

// main statemachine of base controller
CASE me.StateMachine.intState OF
	cSTA_RUNBusy:
		THIS^.sta_RUNBusy();
	cSTA_RUN:
		THIS^.sta_RUN();
	cSTA_STOPBusy: 
        THIS^.sta_STOPBusy();
    cSTA_STOP: 
        THIS^.sta_STOP();
	UMC_CmdState.cSTA_RESETMOTORERROR:
		THIS^.sta_RESETMOTORERROR();
	UMC_CmdState.cSTA_SETOPERATIONMODE:
		THIS^.sta_SETOPERATIONMODE();
END_CASE;
END_METHOD

END_FUNCTION_BLOCK

// POUs/Controller/Lvl0/VLV (Valve controller)/FB_VLV
FUNCTION_BLOCK FB_VLV EXTENDS FB_CtrlBase
VAR_INPUT
	In_bolOpened: BOOL;
	In_bolClosed: BOOL;
END_VAR
VAR_OUTPUT
	Out_bolOpen: BOOL;
	Out_bolClose: BOOL;
END_VAR
VAR
	/// Specific interface struct for public access
	SIf: T_Ctrl_SIf_VLV;
END_VAR

(*__________________________________________________________________________________________________
¦	
¦	Vistaprint Schweiz GmbH
¦	CH - 8401 Winterthur
¦
¦	www.vistaprint.ch - info@vistaprint.ch
¦___________________________________________________________________________________________________

Function desription:
Basic valve controller

History:
Version		Date			Author		Comment
---------------------------------------------------------------------------------------------------
0.00.1		06.03.2014		AVME/DSC	Start history. Based on CYL controller

___________________________________________________________________________________________________*)


IF (me.bolActivate) THEN // cyclic call enabled
	IF (CIf.Info.bolInitDone=FALSE) THEN // first cycle -> init
		CtrlInit();
		CIf.Info.bolInitDone := TRUE;
	ELSE
		CycleStartDuty();
	
		Always();
		
		StateMachine();
		
		CycleEndDuty();
	END_IF
END_IF;

METHOD PROTECTED Always : BOOL
IF (me.bolChangeBackToAUTO=TRUE) THEN // switch mode to automatic switch off controller
	//me.StateMachine.intStateNext := cSTA_OFFBusy;
	me.bolChangeBackToAUTO := FALSE; // for valve no change to off when switch to automatic!!
END_IF

SUPER^.Always();

// ----------------------------------------------------------------------------------
// cyclic actions outside of statemachine
IF (me.StateMachine.intState<>cSTA_SINGLE_ANSWER) THEN
	
	; // always error supervision
	// ----------------------------------------------------------------------------------
	// overrule error always from base -> no EOFF State!! in EOFF go to OFF
	IF (me.StateMachine.intStateNext = cSTA_EOFFBusy) THEN
		IF (me.StateMachine.intState=cSTA_OFF) THEN
			me.StateMachine.intStateNext := cSTA_OFF;
		ELSE // stay in OFF
			me.StateMachine.intStateNext := cSTA_OFFBusy;
		END_IF
	END_IF
END_IF
END_METHOD

METHOD FB_init : BOOL
VAR_INPUT
	///if TRUE, the retain variables are initialized (warm start / cold start)
	bInitRetains: BOOL;
	///if TRUE, the instance afterwards gets moved into the copy code (online change)
	bInCopyCode: BOOL;
END_VAR
VAR
	ii: UINT;
END_VAR
//------------------------------------------------------------------------------------------------------------------------
// to manually change in new FUB implementation!!!
// define valid commands for this controller
FOR ii:= 0 TO (SIZEOF(CIf.Job.aCmdList)/SIZEOF(CIf.Job.aCmdList[0])-1) BY 1 DO
	IF (CIf.Job.aCmdList[ii].intCmd=cCMD_INITIALIZED) THEN
		// found first empty array element
		EXIT;
	END_IF
END_FOR

CIf.Job.aCmdList[ii].intCmd := cCMD_OPEN;
CIf.Job.aCmdList[ii].strName := 'Open';
CIf.Job.aCmdList[ii].bolAvailable := TRUE;
ii := ii +1;
CIf.Job.aCmdList[ii].intCmd := cCMD_CLOSE; 
CIf.Job.aCmdList[ii].strName := 'Close';
CIf.Job.aCmdList[ii].bolAvailable := TRUE;

// set name of class/typ
CIf.Info.strType := 'FB_VLV'; 

// set alarm class
SIf.Alm[E_ALM_VLV.SensorOpenAlwaysOn].eAlmClass := E_AlmClass.TSTOP;
SIf.Alm[E_ALM_VLV.SensorOpenAlwaysOn].strText := 'sensor open always on'; 
SIf.Alm[E_ALM_VLV.SensorOpenNotReached].eAlmClass := E_AlmClass.TSTOP;
SIf.Alm[E_ALM_VLV.SensorOpenNotReached].strText := 'timeout open - sensor open not reached';
SIf.Alm[E_ALM_VLV.SensorCloseAlwaysOn].eAlmClass := E_AlmClass.TSTOP;
SIf.Alm[E_ALM_VLV.SensorCloseAlwaysOn].strText := 'sensor close always on';
SIf.Alm[E_ALM_VLV.SensorCloseNotReached].eAlmClass := E_AlmClass.TSTOP;
SIf.Alm[E_ALM_VLV.SensorCloseNotReached].strText := 'timeout close - sensor close not reached';
SIf.Alm[E_ALM_VLV.InterlockOpen].eAlmClass := E_AlmClass.OFF;
SIf.Alm[E_ALM_VLV.InterlockOpen].strText := 'interlock open - movement stopped';
SIf.Alm[E_ALM_VLV.InterlockClose].eAlmClass := E_AlmClass.OFF;
SIf.Alm[E_ALM_VLV.InterlockClose].strText := 'interlock close - movement stopped';

//*******************************************************************************
// initial values
//*******************************************************************************

// Configuration defaults of class
CIf.SwCfg.bolExist := TRUE;
CIf.SwCfg.bolEnable := TRUE;
CIf.SwCfg.bolSimulation := FALSE;

// Parameter defaults of class
SIf.Par.udiOpenTime_ms := 4000;
SIf.Par.udiCloseTime_ms := 4000;
SIf.Par.udiSimOpenTime_ms := SIf.Par.udiOpenTime_ms/2;	
SIf.Par.udiSimCloseTime_ms := SIf.Par.udiCloseTime_ms/2;
END_METHOD

METHOD PROTECTED getCmdState : STRING
VAR_INPUT
	intCmdState: INT;
	bolState: BOOL;
END_VAR
getCmdState := SUPER^.getCmdState(intCmdState:=intCmdState,bolState:=bolState); // get global/base defined cmds/states
IF (getCmdState='') THEN // global not defined get local
	// get string cmd/state string information in runtime
	IF (bolState=FALSE) THEN
		// cmd's
		CASE intCmdState OF
			VLV_CmdState.cCMD_OPEN: 
				getCmdState := 'cCMD_OPEN';
			VLV_CmdState.cCMD_CLOSE: 
				getCmdState := 'cCMD_CLOSE';
		ELSE
			getCmdState := 'Cmd not defined';
		END_CASE;
	ELSE
	
	// cmd's
		CASE intCmdState OF
			VLV_CmdState.cSTA_OPENBusy: 
				getCmdState := 'cSTA_OPENBusy';
			VLV_CmdState.cSTA_OPEN: 
				getCmdState := 'cSTA_OPEN';
			VLV_CmdState.cSTA_CLOSEBusy: 
				getCmdState := 'cSTA_CLOSEBusy';
			VLV_CmdState.cSTA_CLOSE: 
				getCmdState := 'cSTA_CLOSE';
		ELSE
			getCmdState := 'State not defined';
		END_CASE;
	END_IF
END_IF
END_METHOD

METHOD getCtrlSIf : POINTER TO T_Ctrl_SIf_VLV
getCtrlSIf := ADR(SIf);
END_METHOD

METHOD PROTECTED IoInBridge : BOOL
// digitale and analoge inputs read from hardware or forcing
SIf.In.bolOpen.map := THIS^.In_bolOpened;
SIf.In.bolClose.map := THIS^.In_bolClosed;

IF (CIf.SwCfg.bolSimulation = FALSE) THEN
	getInBol(CIf.Job.bolIoForce,ADR(SIf.In.bolOpen));
	getInBol(CIf.Job.bolIoForce,ADR(SIf.In.bolClose));
ELSE
	//simulation of global IO
END_IF
END_METHOD

METHOD PROTECTED IoOutBridge : BOOL
VAR
	bolSwitchValvesOff: BOOL;
END_VAR
// digitale and analoge inputs read from hardware or forcing
IF (CIf.SwCfg.bolSimulation = FALSE) THEN
	setOutBol(CIf.Job.bolIoForce ,ADR(SIf.Out.bolOpen));
	setOutBol(CIf.Job.bolIoForce ,ADR(SIf.Out.bolClose));
	
	// check interlocks to prevent damages
	IF (CIf.Job.bolIlkOverwrite=FALSE) THEN
		bolSwitchValvesOff := FALSE;
		
		IF (SIf.Ilk.bolOpen=TRUE) THEN
			// switch off?
			IF (SIf.Cfg.eTyp = E_Typ_VLV.Valve1_Sensor0) OR (SIf.Cfg.eTyp = E_Typ_VLV.Valve1_Sensor2) 
				OR (SIf.Cfg.eTyp = E_Typ_VLV.Valve1_SensorOpened) OR (SIf.Cfg.eTyp = E_Typ_VLV.Valve1_SensorClosed) THEN
				// monostabil valve -> do nothing
			ELSE
				// bistable valve ->  switch both off
				bolSwitchValvesOff := TRUE;
				IF (SIf.Out.bolOpen.map=1) THEN
					pfbAlarmCtrl^.setAlarm(CIf.Info.intCtrlId,E_ALM_VLV.InterlockOpen,0,ADR(SIf.Alm),E_AlmState.RST,CIf.Job.eMe_ActivAlmClass);
				END_IF
			END_IF
		END_IF
		
		IF (SIf.Ilk.bolClose=TRUE) THEN
			// switch off?
			IF (SIf.Cfg.eTyp = E_Typ_VLV.Valve1_Sensor0) OR (SIf.Cfg.eTyp = E_Typ_VLV.Valve1_Sensor2) 
				OR (SIf.Cfg.eTyp = E_Typ_VLV.Valve1_SensorOpened) OR (SIf.Cfg.eTyp = E_Typ_VLV.Valve1_SensorClosed) THEN
				// monostabil valve -> do nothing
				;
			ELSE
				// bistable valve -> switch both off
				bolSwitchValvesOff := TRUE;
				IF (SIf.Out.bolClose.map=1) THEN
					pfbAlarmCtrl^.setAlarm(CIf.Info.intCtrlId,E_ALM_VLV.InterlockClose,0,ADR(SIf.Alm),E_AlmState.RST,CIf.Job.eMe_ActivAlmClass);
				END_IF;
			END_IF
		END_IF
		
		// bistable valve -> switch both off
		IF (bolSwitchValvesOff) THEN
			SIf.Out.bolOpen.map := FALSE;
			SIf.Out.bolClose.map := FALSE;
		END_IF
		
	END_IF

	THIS^.Out_bolOpen := SIf.Out.bolOpen.map;
	THIS^.Out_bolClose := SIf.Out.bolClose.map;
END_IF
END_METHOD

METHOD PROTECTED sta_CLOSE : BOOL
// state implemetation
//--------------------------------------------------------------------------------------
// Entry action
	IF (me.StateMachine.intState<>me.StateMachine.intStateLastCycle) THEN
		me.StateMachine.intStateLastCycle := me.StateMachine.intState;

	END_IF

//--------------------------------------------------------------------------------------
// Cyclic action
	IF (me.StateMachine.intState=me.StateMachine.intStateLastCycle) THEN

		// Simulation
		IF (CIf.SwCfg.bolSimulation) THEN
			;
		END_IF
		
		// State Change Condition
		IF (SIf.In.bolOpen.intern) THEN
			// sensor open always on
			pfbAlarmCtrl^.setAlarm(CIf.Info.intCtrlId,E_ALM_VLV.SensorOpenAlwaysOn,0,ADR(SIf.Alm),E_AlmState.RST,CIf.Job.eMe_ActivAlmClass);
			me.StateMachine.intStateNext :=  cSTA_ERROR;
		ELSIF ((SIf.In.bolClose.intern = FALSE) AND ((SIf.Cfg.eTyp = E_Typ_VLV.Valve1_SensorClosed) OR (SIf.Cfg.eTyp = E_Typ_VLV.Valve2_SensorClosed))) THEN // wait time until error?
			me.StateMachine.intStateNext := VLV_CmdState.cSTA_CLOSEBusy;
		ELSIF(me.intCmd=VLV_CmdState.cCMD_OPEN) THEN
			me.StateMachine.intStateNext := VLV_CmdState.cSTA_OPENBusy;
		END_IF
	END_IF

//--------------------------------------------------------------------------------------
// Exit action
	IF (me.StateMachine.intState<>me.StateMachine.intStateNext) THEN
		;
	END_IF
END_METHOD

METHOD PROTECTED sta_CLOSEBusy : BOOL
// state implemetation
//--------------------------------------------------------------------------------------
// Entry action
	IF (me.StateMachine.intState<>me.StateMachine.intStateLastCycle) THEN
		me.StateMachine.intStateLastCycle := me.StateMachine.intState;
		
		SIf.Out.bolOpen.intern := FALSE;
		SIf.Out.bolClose.intern := TRUE;
		
		fbSimulationTimer.IN := FALSE;
		fbSimulationTimer.PT := UDINT_TO_TIME(SIf.Par.udiSimCloseTime_ms);
		fbSimulationTimer(); // set time/reset timer
		fbSimulationTimer.IN := TRUE; // start timer
	END_IF


//--------------------------------------------------------------------------------------
// Cyclic action
	IF (me.StateMachine.intState=me.StateMachine.intStateLastCycle) THEN

		// Simulation
		IF (CIf.SwCfg.bolSimulation) THEN
			fbSimulationTimer(); // simulation time
			IF (fbSimulationTimer.Q) THEN
				SIf.In.bolClose.intern := TRUE;
				SIf.In.bolOpen.intern := FALSE;
			END_IF
		END_IF
		
		// State Change Condition
		IF (me.StateMachine.udiTimeInState_ms>SIf.Par.udiCloseTime_ms) THEN
			IF (SIf.In.bolOpen.intern) THEN
				// sensor open always on 
				pfbAlarmCtrl^.setAlarm(CIf.Info.intCtrlId,E_ALM_VLV.SensorOpenAlwaysOn,0,ADR(SIf.Alm),E_AlmState.RST,CIf.Job.eMe_ActivAlmClass);
			ELSE
				// timeout close valve
				pfbAlarmCtrl^.setAlarm(CIf.Info.intCtrlId,E_ALM_VLV.SensorCloseNotReached,0,ADR(SIf.Alm),E_AlmState.RST,CIf.Job.eMe_ActivAlmClass);
			END_IF
			me.StateMachine.intStateNext :=  cSTA_ERROR;
		ELSIF (SIf.In.bolClose.intern) AND(SIf.In.bolOpen.intern=FALSE) THEN
			me.StateMachine.intStateNext := VLV_CmdState.cSTA_CLOSE;
		ELSIF ((SIf.Cfg.eTyp = E_Typ_VLV.Valve1_SensorOpened) OR (SIf.Cfg.eTyp = E_Typ_VLV.Valve2_SensorOpened))
				 AND (SIf.In.bolOpen.intern=FALSE) AND (me.StateMachine.udiTimeInState_ms>SIf.Par.udiSimCloseTime_ms) THEN
			me.StateMachine.intStateNext := VLV_CmdState.cSTA_CLOSE;
		ELSIF ((SIf.Cfg.eTyp = E_Typ_VLV.Valve1_Sensor0) OR (SIf.Cfg.eTyp = E_Typ_VLV.Valve2_Sensor0))
				AND (me.StateMachine.udiTimeInState_ms>SIf.Par.udiSimCloseTime_ms) THEN
			me.StateMachine.intStateNext := VLV_CmdState.cSTA_CLOSE;		
		ELSIF(me.intCmd=VLV_CmdState.cCMD_OPEN) THEN
			me.StateMachine.intStateNext := VLV_CmdState.cSTA_OPENBusy;
		END_IF
	END_IF


//--------------------------------------------------------------------------------------
// Exit action
	IF (me.StateMachine.intState<>me.StateMachine.intStateNext) THEN
		SIf.Cur.udiMoveTimeClose := me.StateMachine.udiTimeInState_ms;
	END_IF
END_METHOD

METHOD PROTECTED sta_ERROR : BOOL
// state implemetation
//--------------------------------------------------------------------------------------
// Entry action
	IF (me.StateMachine.intState<>me.StateMachine.intStateLastCycle) THEN
		me.StateMachine.intStateHistory := me.StateMachine.intStateLastCycle; // -> possibillity to go back to state before error
		me.StateMachine.intStateLastCycle := me.StateMachine.intState;
		
	END_IF

//--------------------------------------------------------------------------------------
// Cyclic action
	IF (me.StateMachine.intState=me.StateMachine.intStateLastCycle) THEN
		
		;	
		// State Change Condition
		IF (CIf.Job.bolAlmReset = TRUE) THEN
			me.StateMachine.intStateNext := cSTA_ERRORQuit;
		END_IF
	END_IF

//--------------------------------------------------------------------------------------
// Exit action
	IF (me.StateMachine.intState<>me.StateMachine.intStateNext) THEN
		;
	END_IF
END_METHOD

METHOD PROTECTED sta_ERRORQuit : BOOL
// state implemetation
//--------------------------------------------------------------------------------------
// Entry action
	IF (me.StateMachine.intState<>me.StateMachine.intStateLastCycle) THEN
		me.StateMachine.intStateLastCycle := me.StateMachine.intState;
		
	END_IF


//--------------------------------------------------------------------------------------
// Cyclic action
	IF (me.StateMachine.intState=me.StateMachine.intStateLastCycle) THEN
		
		;
		// evtl. wait time if reset of device is necessary and then decide to go to states or ERROR state
		IF (CIf.Job.bolAlmReset = TRUE) THEN
			CIf.Job.eMe_ActivAlmClass := E_AlmClass.NONE; // reset feedback channel for parent
			CIf.Job.bolAlmReset := FALSE;
		END_IF
		
		// State Change Condition
		IF (CIf.Job.bolAlmReset = FALSE) THEN
			IF (me.StateMachine.intStateHistory<=cSTA_PON) THEN
				me.StateMachine.intStateNext := cSTA_PONBusy;
			ELSIF(me.intCmd=cCMD_OFF) THEN
				me.StateMachine.intStateNext := cSTA_OFFBusy;
			ELSIF(me.intCmd=VLV_CmdState.cCMD_OPEN) THEN
				me.StateMachine.intStateNext := VLV_CmdState.cSTA_OPENBusy;
			ELSIF(me.intCmd=VLV_CmdState.cCMD_CLOSE) THEN
				me.StateMachine.intStateNext := VLV_CmdState.cSTA_CLOSEBusy;
			END_IF
		END_IF
	END_IF


//--------------------------------------------------------------------------------------
// Exit action
	IF (me.StateMachine.intState<>me.StateMachine.intStateNext) THEN
		;
	END_IF
END_METHOD

METHOD PROTECTED sta_OFF : BOOL
// state implemetation
//--------------------------------------------------------------------------------------
// Entry action
	IF (me.StateMachine.intState<>me.StateMachine.intStateLastCycle) THEN
		me.StateMachine.intStateLastCycle := me.StateMachine.intState;
		
	END_IF


//--------------------------------------------------------------------------------------
// Cyclic action
	IF (me.StateMachine.intState=me.StateMachine.intStateLastCycle) THEN
		
		;
		
		// State Change Condition
		IF (me.Alarm.eActivAlmClass<>E_AlmClass.EOFF) AND (me.Alarm.eActivAlmClass<>E_AlmClass.OFF) THEN
			IF (me.intCmd=VLV_CmdState.cCMD_OPEN) THEN 
				me.StateMachine.intStateNext := VLV_CmdState.cSTA_OPENBusy;
			ELSIF(me.intCmd=VLV_CmdState.cCMD_CLOSE) THEN
				me.StateMachine.intStateNext := VLV_CmdState.cSTA_CLOSEBusy;
			END_IF
		END_IF
	END_IF




//--------------------------------------------------------------------------------------
// Exit action
	IF (me.StateMachine.intState<>me.StateMachine.intStateNext) THEN
		;
	END_IF
END_METHOD

METHOD PROTECTED sta_OFFBusy : BOOL
// state implemetation
//--------------------------------------------------------------------------------------
// Entry action
	IF (me.StateMachine.intState<>me.StateMachine.intStateLastCycle) THEN
		me.StateMachine.intStateLastCycle := me.StateMachine.intState;
		
	END_IF


//--------------------------------------------------------------------------------------
// Cyclic action
	IF (me.StateMachine.intState=me.StateMachine.intStateLastCycle) THEN
		
		// switch off?
		IF (SIf.Cfg.eTyp = E_Typ_VLV.Valve1_Sensor0) OR (SIf.Cfg.eTyp = E_Typ_VLV.Valve1_Sensor2) 
			OR (SIf.Cfg.eTyp = E_Typ_VLV.Valve1_SensorOpened) OR (SIf.Cfg.eTyp = E_Typ_VLV.Valve1_SensorClosed) THEN
			// monostabil valve -> do nothing
			;
		ELSE
			// bistable valve -> switch both off
			SIf.Out.bolOpen.intern := FALSE;
			SIf.Out.bolClose.intern := FALSE;
		END_IF
		
		
		
		// State Change Condition
		IF (TRUE) THEN
			me.StateMachine.intStateNext := cSTA_OFF;
		END_IF
	END_IF




//--------------------------------------------------------------------------------------
// Exit action
	IF (me.StateMachine.intState<>me.StateMachine.intStateNext) THEN
		;
	END_IF
END_METHOD

METHOD PROTECTED sta_OPEN : BOOL
// state implemetation
//--------------------------------------------------------------------------------------
// Entry action
	IF (me.StateMachine.intState<>me.StateMachine.intStateLastCycle) THEN
		me.StateMachine.intStateLastCycle := me.StateMachine.intState;

	END_IF

//--------------------------------------------------------------------------------------
// Cyclic action
	IF (me.StateMachine.intState=me.StateMachine.intStateLastCycle) THEN

		// Simulation
		IF (CIf.SwCfg.bolSimulation) THEN
			;
		END_IF
		
		// State Change Condition
		IF (SIf.In.bolClose.intern) THEN
			// sensor close always on
			pfbAlarmCtrl^.setAlarm(CIf.Info.intCtrlId,E_ALM_VLV.SensorCloseAlwaysOn,0,ADR(SIf.Alm),E_AlmState.RST,CIf.Job.eMe_ActivAlmClass);
			me.StateMachine.intStateNext :=  cSTA_ERROR;
		ELSIF ((SIf.In.bolOpen.intern = FALSE) AND ((SIf.Cfg.eTyp = E_Typ_VLV.Valve1_SensorOpened) OR (SIf.Cfg.eTyp = E_Typ_VLV.Valve2_SensorOpened))) THEN // wait time until error?
			me.StateMachine.intStateNext := VLV_CmdState.cSTA_OPENBusy;
		ELSIF(me.intCmd=VLV_CmdState.cCMD_CLOSE) THEN
			me.StateMachine.intStateNext := VLV_CmdState.cSTA_CLOSEBusy;
		END_IF
	END_IF

//--------------------------------------------------------------------------------------
// Exit action
	IF (me.StateMachine.intState<>me.StateMachine.intStateNext) THEN
		;
	END_IF
END_METHOD

METHOD PROTECTED sta_OPENBusy : BOOL
// state implemetation
//--------------------------------------------------------------------------------------
// Entry action
	IF (me.StateMachine.intState<>me.StateMachine.intStateLastCycle) THEN
		me.StateMachine.intStateLastCycle := me.StateMachine.intState;

		SIf.Out.bolOpen.intern := TRUE;
		SIf.Out.bolClose.intern := FALSE;
		
		fbSimulationTimer.IN := FALSE;
		fbSimulationTimer.PT := UDINT_TO_TIME(SIf.Par.udiSimOpenTime_ms);
		fbSimulationTimer(); // set time/reset timer
		fbSimulationTimer.IN := TRUE; // start timer
	END_IF


//--------------------------------------------------------------------------------------
// Cyclic action
	IF (me.StateMachine.intState=me.StateMachine.intStateLastCycle) THEN

		// Simulation
		IF (CIf.SwCfg.bolSimulation) THEN
			fbSimulationTimer(); // simulation time
			IF (fbSimulationTimer.Q) THEN
				SIf.In.bolOpen.intern := TRUE;
				SIf.In.bolClose.intern := FALSE;
			END_IF
		END_IF
		
		// State Change Condition
		IF (me.StateMachine.udiTimeInState_ms > SIf.Par.udiOpenTime_ms) THEN
			IF (SIf.In.bolClose.intern) THEN
				// sensor close always on
				pfbAlarmCtrl^.setAlarm(CIf.Info.intCtrlId,E_ALM_VLV.SensorCloseAlwaysOn,0,ADR(SIf.Alm),E_AlmState.RST,CIf.Job.eMe_ActivAlmClass);
			ELSE
				// timeout open valve
				pfbAlarmCtrl^.setAlarm(CIf.Info.intCtrlId,E_ALM_VLV.SensorOpenNotReached,0,ADR(SIf.Alm),E_AlmState.RST,CIf.Job.eMe_ActivAlmClass);
			END_IF
			me.StateMachine.intStateNext :=  cSTA_ERROR;
		ELSIF (SIf.In.bolOpen.intern) AND (SIf.In.bolClose.intern=FALSE) THEN
			me.StateMachine.intStateNext := VLV_CmdState.cSTA_OPEN;
		ELSIF ((SIf.Cfg.eTyp = E_Typ_VLV.Valve1_SensorClosed) OR (SIf.Cfg.eTyp = E_Typ_VLV.Valve2_SensorClosed))
				 AND (SIf.In.bolClose.intern=FALSE) AND (me.StateMachine.udiTimeInState_ms>SIf.Par.udiSimOpenTime_ms) THEN
			me.StateMachine.intStateNext := VLV_CmdState.cSTA_OPEN;
		ELSIF ((SIf.Cfg.eTyp = E_Typ_VLV.Valve1_Sensor0) OR (SIf.Cfg.eTyp = E_Typ_VLV.Valve2_Sensor0))
				AND (me.StateMachine.udiTimeInState_ms>SIf.Par.udiSimOpenTime_ms) THEN
			me.StateMachine.intStateNext := VLV_CmdState.cSTA_OPEN;		
		ELSIF(me.intCmd=VLV_CmdState.cCMD_CLOSE) THEN
			me.StateMachine.intStateNext := VLV_CmdState.cSTA_CLOSEBusy;
		END_IF
	END_IF

//--------------------------------------------------------------------------------------
// Exit action
	IF (me.StateMachine.intState<>me.StateMachine.intStateNext) THEN
		SIf.Cur.udiMoveTimeOpen := me.StateMachine.udiTimeInState_ms;
	END_IF
END_METHOD

METHOD PROTECTED StateMachine : BOOL
SUPER^.StateMachine();

// main statemachine of base controller
CASE me.StateMachine.intState OF
    VLV_CmdState.cSTA_OPENBusy: 
        THIS^.sta_OPENBusy();
    VLV_CmdState.cSTA_OPEN: 
        THIS^.sta_OPEN();
    VLV_CmdState.cSTA_CLOSEBusy: 
        THIS^.sta_CLOSEBusy();
    VLV_CmdState.cSTA_CLOSE: 
        THIS^.sta_CLOSE();
END_CASE;
END_METHOD

END_FUNCTION_BLOCK

// POUs/Controller/Lvl0/VPC [Vacuum Pump Controller]/FB_VPC
FUNCTION_BLOCK FB_VPC EXTENDS FB_CtrlBase
VAR_INPUT
	In_bolVacuumOk			: BOOL;
	In_bolPumpOk			: BOOL;
END_VAR
VAR_OUTPUT
	Out_bolVaccumPumpOn		: BOOL;
END_VAR
VAR
	/// Specific interface struct for public access
	SIf					: T_Ctrl_SIf_VPC;
END_VAR

(*__________________________________________________________________________________________________
¦	
¦	Vistaprint Schweiz GmbH
¦	CH - 8401 Winterthur
¦
¦	www.vistaprint.ch - info@vistaprint.ch
¦___________________________________________________________________________________________________

Function desription:
Vacuum Pump implementation. 


History:
Version		Date			Author		Comment
---------------------------------------------------------------------------------------------------
0.00.1		09.07.2013		PC			Start history
___________________________________________________________________________________________________*)


IF (me.bolActivate) THEN // cyclic call enabled
	IF (CIf.Info.bolInitDone=FALSE) THEN // first cycle -> init
		CtrlInit();
		CIf.Info.bolInitDone := TRUE;
	ELSE
		CycleStartDuty();
	
		Always();
		
		StateMachine();
		
		CycleEndDuty();
	END_IF
END_IF;

METHOD PROTECTED Always : BOOL
SUPER^.Always();

// ----------------------------------------------------------------------------------
// cyclic actions outside of statemachine
IF (me.StateMachine.intState<>cSTA_SINGLE_ANSWER) THEN
	
	; // always error supervision
	
END_IF

// ----------------------------------------------------------------------------------
// Conditions Always
IF (((me.Alarm.eActivAlmClass=E_AlmClass.EOFF) OR (me.Alarm.eActivAlmClass=E_AlmClass.OFF) OR (me.intCmd=cCMD_OFF))
		 AND (me.StateMachine.intState<>cSTA_ERROR) AND (me.StateMachine.intState<>cSTA_ERRORQuit) AND
		(me.StateMachine.intState<>cSTA_OFF) AND (me.StateMachine.intState<>cSTA_OFFBusy)) THEN
	// alarm evt EOFF, OFF or cmd off
	me.StateMachine.intStateNext := cSTA_OFFBusy;
END_IF
END_METHOD

METHOD FB_init : BOOL
VAR_INPUT
	bInitRetains : BOOL; // if TRUE, the retain variables are initialized (warm start / cold start)
	bInCopyCode : BOOL;  // if TRUE, the instance afterwards gets moved into the copy code (online change)
END_VAR
VAR
	iIdx		: UINT;
	iLength		: UINT;	
END_VAR
//------------------------------------------------------------------------------------------------------------------------
// to manually change in new FUB implementation!!!
// define valid commands for this controller
iLength := SIZEOF(CIf.Job.aCmdList)/SIZEOF(CIf.Job.aCmdList[0]);
iIdx := 0;

WHILE (iIdx < iLength) AND (CIf.Job.aCmdList[iIdx].intCmd <> cCMD_INITIALIZED) DO
	iIdx := iIdx + 1; 
END_WHILE

IF (iIdx < iLength) THEN
// Add configuration of own comands	
	CIf.Job.aCmdList[iIdx].intCmd := BASE_PLC.cCMD_RUN;
	CIf.Job.aCmdList[iIdx].strName := 'RUN'; 
	CIf.Job.aCmdList[iIdx].bolAvailable := TRUE;
ELSE
	// Error if the aCmdList Array is to small
END_IF

// set name of class/typ
CIf.Info.strType := 'FB_VPC'; 

// set alarm class
SIf.Alm[E_ALM_VPC.VacuumPumpOnTimeout].eAlmClass := E_AlmClass.TSTOP;
SIf.Alm[E_ALM_VPC.VacuumPumpOnTimeout].strText := 'Vacuum pump On timeout'; 
SIf.Alm[E_ALM_VPC.VacuumPumpOffTimeout].eAlmClass := E_AlmClass.TSTOP;
SIf.Alm[E_ALM_VPC.VacuumPumpOffTimeout].strText := 'Vacuum pump Off timeout';
SIf.Alm[E_ALM_VPC.VacuumFailure].eAlmClass := E_AlmClass.TSTOP;
SIf.Alm[E_ALM_VPC.VacuumFailure].strText := 'Vacuum failure';

//*******************************************************************************
// initial values
//*******************************************************************************

// software configuration
CIf.SwCfg.bolExist := TRUE;
CIf.SwCfg.bolEnable := TRUE;
CIf.SwCfg.bolSimulation := FALSE;

// parameter
SIf.Par.udiVacuumPumpTime_ms := 10000;
SIf.Par.udiVacuumStabilizationTime_ms := 3000;
SIf.Par.udiSimVacuumPumpOnTime_ms := SIf.Par.udiVacuumPumpTime_ms / 2;
END_METHOD

METHOD PROTECTED getCmdState : STRING

VAR_INPUT
	intCmdState: INT;
	bolState: BOOL;
END_VAR
getCmdState := SUPER^.getCmdState(intCmdState:=intCmdState,bolState:=bolState); // get global/base defined cmds/states

IF (getCmdState='') THEN // global not defined get local
	// get string cmd/state string information in runtime
	IF (bolState=FALSE) THEN
		;// Comands's
	ELSE
		// States's
		CASE intCmdState OF
			VPC_CmdState.cSTA_VPC_StabilizeBusy: 
				getCmdState := 'cSTA_StabilizeBusy';
		END_CASE;
	END_IF
END_IF
END_METHOD

METHOD getCtrlSIf : POINTER TO T_Ctrl_SIf_VPC
getCtrlSIf := ADR(SIf);
END_METHOD

METHOD PROTECTED IoInBridge : BOOL
// digitale and analoge inputs read from hardware or forcing
SIf.In.bolVacuumOk.map := THIS^.In_bolVacuumOk;
SIf.In.bolPumpOn.map := THIS^.In_bolPumpOk;

IF (CIf.SwCfg.bolSimulation = FALSE) THEN
	getInBol(CIf.Job.bolIoForce,ADR(SIf.In.bolVacuumOk));
	getInBol(CIf.Job.bolIoForce,ADR(SIf.In.bolPumpOn));
ELSE
	//simulation of global IO
END_IF
END_METHOD

METHOD PROTECTED IoOutBridge : BOOL
VAR
	bolSwitchValvesOff: BOOL;
END_VAR
// digitale and analoge inputs read from hardware or forcing
IF (CIf.SwCfg.bolSimulation = FALSE) THEN
	setOutBol(CIf.Job.bolIoForce ,ADR(SIf.Out.bolVacuumPumpOn));

	THIS^.Out_bolVaccumPumpOn := SIf.Out.bolVacuumPumpOn.map;
END_IF
END_METHOD

METHOD PROTECTED sta_ERROR : BOOL
// state implemetation
//--------------------------------------------------------------------------------------
// Entry action
	IF (me.StateMachine.intState<>me.StateMachine.intStateLastCycle) THEN
		me.StateMachine.intStateHistory := me.StateMachine.intStateLastCycle; // -> possibillity to go back to state before error
		me.StateMachine.intStateLastCycle := me.StateMachine.intState;
		
	END_IF


//--------------------------------------------------------------------------------------
// Cyclic action
	IF (me.StateMachine.intState=me.StateMachine.intStateLastCycle) THEN
		
		;
		
		
		// State Change Condition
		IF (CIf.Job.bolAlmReset = TRUE) THEN
			me.StateMachine.intStateNext := cSTA_ERRORQuit;
		END_IF
	END_IF




//--------------------------------------------------------------------------------------
// Exit action
	IF (me.StateMachine.intState<>me.StateMachine.intStateNext) THEN
		;
	END_IF
END_METHOD

METHOD PROTECTED sta_ERRORQuit : BOOL
// state implemetation
//--------------------------------------------------------------------------------------
// Entry action
	IF (me.StateMachine.intState<>me.StateMachine.intStateLastCycle) THEN
		me.StateMachine.intStateLastCycle := me.StateMachine.intState;
		
	END_IF


//--------------------------------------------------------------------------------------
// Cyclic action
	IF (me.StateMachine.intState=me.StateMachine.intStateLastCycle) THEN
		
		;
		// evtl. wait time if reset of device is necessary and then decide to go to states or ERROR state
		IF (CIf.Job.bolAlmReset = TRUE) THEN
			CIf.Job.eMe_ActivAlmClass := E_AlmClass.NONE; // reset feedback channel for parent
			CIf.Job.bolAlmReset := FALSE;
		END_IF
		
		// State Change Condition
		IF (CIf.Job.bolAlmReset = FALSE) THEN
			IF (me.StateMachine.intStateHistory<=cSTA_PON) THEN
				me.StateMachine.intStateNext := cSTA_PONBusy;
			ELSIF(me.intCmd=cCMD_OFF) THEN
				me.StateMachine.intStateNext := cSTA_OFFBusy;
			ELSIF(me.intCmd=cCMD_STOP) THEN
				me.StateMachine.intStateNext := cSTA_STOPBusy;
			ELSIF(me.intCmd=BASE_PLC.cCMD_RUN) THEN
				me.StateMachine.intStateNext := BASE_PLC.cSTA_RUNBusy;
			END_IF
		END_IF
	END_IF




//--------------------------------------------------------------------------------------
// Exit action
	IF (me.StateMachine.intState<>me.StateMachine.intStateNext) THEN
		;
	END_IF
END_METHOD

METHOD PROTECTED sta_OFF : BOOL
VAR_INPUT
END_VAR
// state implemetation
//--------------------------------------------------------------------------------------
// Entry action
	IF (me.StateMachine.intState<>me.StateMachine.intStateLastCycle) THEN
		me.StateMachine.intStateLastCycle := me.StateMachine.intState;

	END_IF


//--------------------------------------------------------------------------------------
// Cyclic action
	IF (me.StateMachine.intState=me.StateMachine.intStateLastCycle) THEN
		IF me.intCmd = BASE_PLC.cCMD_RUN THEN
			me.StateMachine.intStateNext := BASE_PLC.cSTA_RUNBusy;
		END_IF
	END_IF


//--------------------------------------------------------------------------------------
// Exit action
	IF (me.StateMachine.intState<>me.StateMachine.intStateNext) THEN
		;
	END_IF
END_METHOD

METHOD PROTECTED sta_OFFBusy : BOOL
VAR_INPUT
END_VAR
// state implemetation
//--------------------------------------------------------------------------------------
// Entry action
	IF (me.StateMachine.intState<>me.StateMachine.intStateLastCycle) THEN
		me.StateMachine.intStateLastCycle := me.StateMachine.intState;
		// Switch Pump Off
		SIf.Out.bolVacuumPumpOn.intern := FALSE;
	END_IF


//--------------------------------------------------------------------------------------
// Cyclic action
	IF (me.StateMachine.intState=me.StateMachine.intStateLastCycle) THEN
		IF (CIf.SwCfg.bolSimulation) THEN
			SIf.In.bolPumpOn.intern := FALSE;
			SIf.In.bolVacuumOk.intern := FALSE;
		END_IF

		IF ((NOT SIf.In.bolPumpOn.intern) OR (NOT SIf.Cfg.VacuumPumpFeedback)) AND ((NOT SIf.In.bolVacuumOk.intern) OR (NOT SIf.Cfg.VacuumSensorAvailable)) THEN
			me.StateMachine.intStateNext := BASE_PLC.cSTA_OFF;
		END_IF;	
	END_IF


//--------------------------------------------------------------------------------------
// Exit action
	IF (me.StateMachine.intState<>me.StateMachine.intStateNext) THEN
		;
	END_IF
END_METHOD

METHOD PROTECTED sta_PON : BOOL
VAR_INPUT
END_VAR
// state implemetation
//--------------------------------------------------------------------------------------
// Entry action
	IF (me.StateMachine.intState<>me.StateMachine.intStateLastCycle) THEN
		me.StateMachine.intStateLastCycle := me.StateMachine.intState;
		
	END_IF


//--------------------------------------------------------------------------------------
// Cyclic action
	IF (me.StateMachine.intState=me.StateMachine.intStateLastCycle) THEN
		;
	END_IF




//--------------------------------------------------------------------------------------
// Exit action
	IF (me.StateMachine.intState<>me.StateMachine.intStateNext) THEN
		;
	END_IF
END_METHOD

METHOD PROTECTED sta_RUN : BOOL
VAR_INPUT
END_VAR
// state implemetation
//--------------------------------------------------------------------------------------
// Entry action
	IF (me.StateMachine.intState<>me.StateMachine.intStateLastCycle) THEN
		me.StateMachine.intStateLastCycle := me.StateMachine.intState;
	END_IF


//--------------------------------------------------------------------------------------
// Cyclic action
	IF (me.StateMachine.intState=me.StateMachine.intStateLastCycle) THEN
		// State Change Condition
		IF (NOT SIf.In.bolPumpOn.intern) AND (SIf.Cfg.VacuumPumpFeedback) THEN
			pfbAlarmCtrl^.setAlarm(CIf.Info.intCtrlId,INT_TO_UINT(E_ALM_VPC.VacuumPumpOnTimeout),0,ADR(SIf.Alm),E_AlmState.RST,CIf.Job.eMe_ActivAlmClass);
			me.StateMachine.intStateNext :=  BASE_PLC.cSTA_ERROR;
		END_IF;

		IF ((NOT SIf.In.bolVacuumOk.intern) AND (SIf.Cfg.VacuumSensorAvailable)) THEN
			pfbAlarmCtrl^.setAlarm(CIf.Info.intCtrlId,INT_TO_UINT(E_ALM_VPC.VacuumFailure),0,ADR(SIf.Alm),E_AlmState.RST,CIf.Job.eMe_ActivAlmClass);
			me.StateMachine.intStateNext :=  BASE_PLC.cSTA_ERROR;
		END_IF;	
	END_IF


//--------------------------------------------------------------------------------------
// Exit action
	IF (me.StateMachine.intState<>me.StateMachine.intStateNext) THEN
		;
	END_IF
END_METHOD

METHOD PROTECTED sta_RUNBusy : BOOL
VAR_INPUT
END_VAR
// state implemetation
//--------------------------------------------------------------------------------------
// Entry action
	IF (me.StateMachine.intState<>me.StateMachine.intStateLastCycle) THEN
		me.StateMachine.intStateLastCycle := me.StateMachine.intState;
		SIf.Out.bolVacuumPumpOn.intern := TRUE;

		fbSimulationTimer.IN := FALSE;
		fbSimulationTimer.PT := UDINT_TO_TIME(SIf.Par.udiSimVacuumPumpOnTime_ms);
		fbSimulationTimer(); // set time/reset timer
		fbSimulationTimer.IN := TRUE; // start timer
	END_IF


//--------------------------------------------------------------------------------------
// Cyclic action
	IF (me.StateMachine.intState=me.StateMachine.intStateLastCycle) THEN
		// Simulation
		IF (CIf.SwCfg.bolSimulation) THEN
			fbSimulationTimer(); // simulation time
			IF (fbSimulationTimer.Q) THEN
				SIf.In.bolPumpOn.intern := TRUE;
				SIf.In.bolVacuumOk.intern := TRUE;
			END_IF
		END_IF

		IF ((SIf.In.bolVacuumOk.intern) OR (NOT SIf.Cfg.VacuumPumpFeedback)) AND ((SIf.In.bolVacuumOk.intern) OR (NOT SIf.Cfg.VacuumSensorAvailable)) THEN
			me.StateMachine.intStateNext := VPC_CmdState.cSTA_VPC_StabilizeBusy;
		END_IF;		
		
		IF (me.StateMachine.udiTimeInState_ms > SIf.Par.udiVacuumPumpTime_ms) THEN
			IF (NOT SIf.In.bolPumpOn.intern) AND (SIf.Cfg.VacuumPumpFeedback) THEN
				pfbAlarmCtrl^.setAlarm(CIf.Info.intCtrlId,INT_TO_UINT(E_ALM_VPC.VacuumPumpOnTimeout),0,ADR(SIf.Alm),E_AlmState.RST,CIf.Job.eMe_ActivAlmClass);
			END_IF;

			IF ((NOT SIf.In.bolVacuumOk.intern) AND (SIf.Cfg.VacuumSensorAvailable)) THEN
				pfbAlarmCtrl^.setAlarm(CIf.Info.intCtrlId,INT_TO_UINT(E_ALM_VPC.VacuumFailure),0,ADR(SIf.Alm),E_AlmState.RST,CIf.Job.eMe_ActivAlmClass);
			END_IF;	

			me.StateMachine.intStateNext :=  cSTA_ERROR;
		END_IF
	END_IF


//--------------------------------------------------------------------------------------
// Exit action
	IF (me.StateMachine.intState<>me.StateMachine.intStateNext) THEN
		;
	END_IF
END_METHOD

METHOD PROTECTED sta_StabilizeVacuum : BOOL
VAR_INPUT
END_VAR
// state implemetation
//--------------------------------------------------------------------------------------
// Entry action
	IF (me.StateMachine.intState<>me.StateMachine.intStateLastCycle) THEN
		me.StateMachine.intStateLastCycle := me.StateMachine.intState;
	END_IF


//--------------------------------------------------------------------------------------
// Cyclic action
	IF (me.StateMachine.intState=me.StateMachine.intStateLastCycle) THEN
		// State Change Condition
		
		IF (me.StateMachine.udiTimeInState_ms > SIf.Par.udiVacuumStabilizationTime_ms) THEN
			me.StateMachine.intStateNext :=  BASE_PLC.cSTA_RUN;
		END_IF;	

		IF (NOT SIf.In.bolPumpOn.intern) AND (SIf.Cfg.VacuumPumpFeedback) THEN
			pfbAlarmCtrl^.setAlarm(CIf.Info.intCtrlId,INT_TO_UINT(E_ALM_VPC.VacuumPumpOnTimeout),0,ADR(SIf.Alm),E_AlmState.RST,CIf.Job.eMe_ActivAlmClass);
			me.StateMachine.intStateNext :=  BASE_PLC.cSTA_ERROR;
		END_IF;

		IF ((NOT SIf.In.bolVacuumOk.intern) AND (SIf.Cfg.VacuumSensorAvailable)) THEN
			pfbAlarmCtrl^.setAlarm(CIf.Info.intCtrlId,INT_TO_UINT(E_ALM_VPC.VacuumFailure),0,ADR(SIf.Alm),E_AlmState.RST,CIf.Job.eMe_ActivAlmClass);
			me.StateMachine.intStateNext :=  BASE_PLC.cSTA_ERROR;
		END_IF;	
	END_IF


//--------------------------------------------------------------------------------------
// Exit action
	IF (me.StateMachine.intState<>me.StateMachine.intStateNext) THEN
		;
	END_IF
END_METHOD

METHOD PROTECTED StateMachine : BOOL
SUPER^.StateMachine();

// main statemachine of base controller
CASE me.StateMachine.intState OF
    VPC_CmdState.cSTA_VPC_StabilizeBusy: 
        THIS^.sta_StabilizeVacuum();
	cSTA_RUNBusy: 
        THIS^.sta_RUNBusy();
    cSTA_RUN: 
        THIS^.sta_RUN();
END_CASE;
END_METHOD

END_FUNCTION_BLOCK

// POUs/Controller/Lvl3/BaseCtrlModule/FB_CtrlModule
FUNCTION_BLOCK FB_CtrlModule EXTENDS FB_CtrlBase
VAR_INPUT
	/// Inputs from global module for general supervision 
	/// Emergency circuit ok
	In_bolEmergencyOffOk: BOOL;
	/// No general error active, will be set to FALSE if there is an global error like e.g. over temperature in cabinet. 
	In_bolNoGeneralError: BOOL;
END_VAR
VAR
	/// Timeout supervision of Keep alive Toggle Bit
	udinTimeToggle_ms: UDINT;
	/// Specific interface struct
	SIf_MOD: T_Ctrl_SIf_MOD;
	uinGroupIndex: UINT;
	intCheckCounter: INT;
	uinMaxNrOfGroups: UINT := Base_Const.cMaxNrOfChilds;
	/// List of sequences
	aListOfSeq: ARRAY[0..Base_Const.cMaxNrOfChilds] OF T_Sequence;
	usiNumOfSeq: USINT := 0;
	usiNumOfValidPointerSeqChild: USINT := 0;
	/// [ms] List of waiting times for run sequence until the next group will execute
	/// If wait time is zero, next group will be directly executed after current group.  
	///	aListOfRunGrpWaitTime_ms: ARRAY[0..Base_Const.cMaxNrOfChilds] OF UDINT;
	usiNumOfRunGrpWaitTime: USINT := 0;
	/// [ms] List of waiting times for stop sequence until the next group will execute
	/// If wait time is zero, next group will be directly executed after current group. 
	///	aListOfStopGrpWaitTime_ms: ARRAY[0..Base_Const.cMaxNrOfChilds] OF UDINT;
	usiNumOfStopGrpWaitTime: USINT := 0;
	/// Array includes all registered childs of type IBuffer
	a_IBufferChildCtrl: ARRAY[0..Base_Const.cMaxNrOfChilds] OF IBuffer;
	a_IBufferFullChildCtrl: ARRAY[0..Base_Const.cMaxNrOfChilds] OF IBuffer;
	usiNumOfIBufferChild: USINT;
	usiNumOfIBufferFullChild: USINT;
	/// Counter
	ii: INT;
END_VAR
VAR CONSTANT
	/// sub States for run and stop sequences
	cSTA_SUB_INITIALIZED: INT := 500;
	cSTA_SUB_SEND_GROUP_CMD: INT := 502;
	cSTA_SUB_CHECK_GROUP_STATUS: INT := 504;
	cSTA_SUB_WAIT: INT := 506;
	cSTA_SUB_FINISHED: INT := 508;
END_VAR

(*__________________________________________________________________________________________________
¦	
¦	Vistaprint Schweiz GmbH
¦	CH - 8401 Winterthur
¦
¦	www.vistaprint.ch - info@vistaprint.ch
¦___________________________________________________________________________________________________

Function desription:
Basic module controller implementation. This Controller should be the base father controller for all modules in shirt stream. 
e.g. used for ICL, ICB, Loading ...

Controller handle following basic functions:
--------------------------------------------
- Monitoring of common signals from cabinet
- Keep alive bit to line control
- General child handling RUN_busy, STOP_busy sequences and error handling

History:
Version		Date			Author		Comment
---------------------------------------------------------------------------------------------------
0.00.1		06.11.2013		AVM/DSC		Start history
0.00.2		14.11.2013		AVM/MRU		Changes in some methods
0.00.3		29.11.2013		AVM/MRU		Changes in IoInBridge
0.00.4		04.12.2013		AVM/MRU		Changes in Always - EOFFBusy
0.00.5		04.12.2013		AVM/MRU		Changes in Always - EOFFBusy at GeneralError
0.00.6		04.12.2013		AVM/MRU		Changes in Always - EOFFBusy if not in sta_EOFF 
0.00.7		05.12.2013		AVM/DSC		General revision of behaviour in case of emergency off (state EOFF) and general error (state ERROR).
										New handling for module specific interface.
0.00.8		06.12.2013		AVM/MRU		Add TSTOP in checkChildAlmClass
0.00.9		09.12.2013		AVM/DSC		BugFix in sub state "cSTA_SUB_CHECK_GROUP_STATUS" from run and stop sequence. Insert new "bolChecked" flag
						 				to detect if the sequence has been processed correctly.
0.00.10		11.12.2013		AVM/MRU		Clear pending command to prevent automatic recovery in sta_STOPBusy
0.00.11		13.01.2014		AVM/MRU		Bugzilla ID 03: BufferFull added
0.00.12		20.01.2014		AVM/MRU		EMO, general error reworked; AddRunGrp, AddStopGrp removed
										Timeout run/stop group added 
0.00.13		22.01.2014		AVM/MRU		Alternativ status for run sequence added
0.00.14		08.02.2014		VP/RE		Added bolStopReleaseHangers to CUR.

___________________________________________________________________________________________________*)


IF (me.bolActivate) AND (SIf_MOD.Cur<>0) AND (SIf_MOD.Cfg<>0) AND (SIf_MOD.Par<>0) AND (SIf_MOD.In<>0) THEN // cyclic call enabled
	IF (CIf.Info.bolInitDone=FALSE) THEN // first cycle -> init
		CtrlInit();
		CIf.Info.bolInitDone := TRUE;
	ELSE
		CycleStartDuty();

		Always();
		
		StateMachine();
		
		CycleEndDuty();
	END_IF
END_IF;

METHOD AddIBufferChilds
VAR_INPUT
	pFB_ChildTypeIBuffer: POINTER TO FB_IBuffer;
END_VAR
// Method add childs with type of IBuffer to the array
IF (usiNumOfIBufferChild <= (Base_Const.cMaxNrOfChilds-1)) THEN
	// Add child controller to list
	a_IBufferChildCtrl[usiNumOfIBufferChild] := pFB_ChildTypeIBuffer^;
	// Inc. number of IBuffer childs
	usiNumOfIBufferChild:= usiNumOfIBufferChild+1;
END_IF
END_METHOD

METHOD AddIBufferFullChilds
VAR_INPUT
	pFB_ChildTypeIBuffer: POINTER TO FB_IBuffer;
END_VAR
// Method add childs with BufferFull information to the array
IF (usiNumOfIBufferFullChild <= (Base_Const.cMaxNrOfChilds-1)) THEN
	// Add child controller to list
	a_IBufferFullChildCtrl[usiNumOfIBufferFullChild] := pFB_ChildTypeIBuffer^;

	// Inc. number of IBufferFull childs
	usiNumOfIBufferFullChild:= usiNumOfIBufferFullChild+1;
END_IF
END_METHOD

METHOD AddSeqChild
VAR_INPUT
	stSequence: T_Sequence;
END_VAR
// Method add a sequence to list
IF (usiNumOfSeq <= (Base_Const.cMaxNrOfChilds-1)) THEN
	aListOfSeq[usiNumOfSeq].pChild:= stSequence.pChild;
	aListOfSeq[usiNumOfSeq].uinGroupRun:= stSequence.uinGroupRun;
	aListOfSeq[usiNumOfSeq].uinGroupStop:= stSequence.uinGroupStop;
	aListOfSeq[usiNumOfSeq].intCmdSeqRun:= stSequence.intCmdSeqRun;
	aListOfSeq[usiNumOfSeq].intStatusSeqRun:= stSequence.intStatusSeqRun;
	aListOfSeq[usiNumOfSeq].intStatusSeqRun2:= stSequence.intStatusSeqRun2;
	aListOfSeq[usiNumOfSeq].intCmdSeqStop:= stSequence.intCmdSeqStop;
	aListOfSeq[usiNumOfSeq].intStatusSeqStop:= stSequence.intStatusSeqStop;
	// Inc. number of sequence
	usiNumOfSeq:= usiNumOfSeq+1;
	// Check if the pointer is valid
	IF (stSequence.pChild<>0) THEN
		usiNumOfValidPointerSeqChild:= usiNumOfValidPointerSeqChild+1;
	END_IF
END_IF
END_METHOD

METHOD PROTECTED Always : BOOL
SUPER^.Always();

// ---------------------------------------------------------------------------------
// Simulation
IF (CIf.SwCfg.bolSimulation) THEN
	SIf_Cur^.bolKeepAliveHost := NOT SIf_Cur^.bolKeepAlivePlc;
	// Simulate inputs from global module for general supervision (no physical inputs)
	SIf_In^.bolEmergencyOffOK.intern := TRUE;
	SIf_In^.bolNoGeneralError.intern := TRUE;
END_IF

// ----------------------------------------------------------------------------------
// cyclic actions outside of statemachine
IF (me.StateMachine.intState<>cSTA_SINGLE_ANSWER) THEN
	
	//-------------------------------------------------------------------------------
	// Monitoring of inputs from global module (no physical inputs)
	//-------------------------------------------------------------------------------
	
	// No general error
	IF ((SIf_In^.bolNoGeneralError.intern = FALSE) AND (me.StateMachine.intState <> cSTA_ERROR) AND (me.StateMachine.intState <> cSTA_ERRORQuit) 
		AND (me.StateMachine.intState <> cSTA_EOFF) AND (me.StateMachine.intState <> cSTA_EOFFBusy)) THEN
		me.StateMachine.intStateNext := cSTA_Error;		
	END_IF
	// As long as general error is not OK, set Alarm
	IF (SIf_In^.bolNoGeneralError.intern = FALSE) AND (me.StateMachine.intState = BASE_PLC.cSTA_ERROR) THEN
		// Set Alarm: SIf_MOD.Alm[4].strText := 'General error active'; 
		pfbAlarmCtrl^.setAlarm(CIf.Info.intCtrlId,4,0,ADR(SIf_MOD.Alm),E_AlmState.RST,CIf.Job.eMe_ActivAlmClass);		
	END_IF
	
	// Emergency Off
	IF ((SIf_In^.bolEmergencyOffOk.intern = FALSE) AND (me.StateMachine.intState <> cSTA_EOFF) AND (me.StateMachine.intState <> cSTA_EOFFBusy)
		AND (me.StateMachine.intState <> cSTA_ERROR) AND (me.StateMachine.intState <> cSTA_ERRORQuit)) THEN
		me.StateMachine.intStateNext := cSTA_EOFFBusy;				
	END_IF
	// As long as EMO is not OK, set Alarm
	IF (SIf_In^.bolEmergencyOffOk.intern = FALSE) AND ((me.StateMachine.intState = cSTA_EOFF) OR (me.StateMachine.intState = cSTA_EOFFBusy)) THEN
		// Set Alarm: SIf_MOD.Alm[3].strText := 'Emergency off active'; 
		pfbAlarmCtrl^.setAlarm(CIf.Info.intCtrlId,3,0,ADR(SIf_MOD.Alm),E_AlmState.RST,CIf.Job.eMe_ActivAlmClass);				
	END_IF
	
END_IF

//-------------------------------------------------------------------------------
// Keep Alive function to line controller with togglebit
//-------------------------------------------------------------------------------

// Communication to line control enabled
IF (SIf_Cfg^.bolComToLineControlEnabled = TRUE) THEN
	IF (SIf_Cur^.bolKeepAliveHost <> SIf_Cur^.bolKeepAlivePlc) THEN
		udinTimeToggle_ms := 0;
		SIf_Cur^.bolKeepAlivePlc := SIf_Cur^.bolKeepAliveHost;
	ELSE
		IF (udinTimeToggle_ms >= SIf_Par^.udiComTimeOutLineCtrl_ms) THEN
			// Set Alarm: SIf_MOD.Alm[2].strText := 'Communication error to line control'; 
			pfbAlarmCtrl^.setAlarm(CIf.Info.intCtrlId,2,UDINT_TO_DINT(udinTimeToggle_ms),ADR(SIf_MOD.Alm),E_AlmState.RST,CIf.Job.eMe_ActivAlmClass);	
			me.StateMachine.intStateNext := cSTA_Error;	
		END_IF
		udinTimeToggle_ms:= udinTimeToggle_ms + me.FUBInfo.udiSample_ms;
	END_IF
// Communication to line control disabled
ELSE
	SIf_Cur^.bolKeepAliveHost:= NOT SIf_Cur^.bolKeepAlivePlc;
END_IF

//-------------------------------------------------------------------------------
// Calculate the sum of all hangers in the system and the capacity of the system
//-------------------------------------------------------------------------------
IF (usiNumOfIBufferChild>0) THEN 
	SIf_Cur^.dinNumOfHangers:= 0;
	SIf_Cur^.dinMaxCapacity:= 0;
	FOR ii:= 0 TO (usiNumOfIBufferChild-1) DO
		SIf_Cur^.dinNumOfHangers:= SIf_Cur^.dinNumOfHangers + a_IBufferChildCtrl[ii].NumOfHangers;
		SIf_Cur^.dinMaxCapacity:= SIf_Cur^.dinMaxCapacity + a_IBufferChildCtrl[ii].MaxCapacity;
	END_FOR
END_IF

//-------------------------------------------------------------------------------
// Write BufferFull for LineControl into SIF
//-------------------------------------------------------------------------------
IF (usiNumOfIBufferFullChild>0) THEN 
	FOR ii:= 0 TO (usiNumOfIBufferFullChild-1) DO
		SIf_Cur^.a_bBufferIsFull[ii]:= a_IBufferFullChildCtrl[ii].BufferFull;
	END_FOR
END_IF


// ----------------------------------------------------------------------------------
// Conditions Always

// EOFF exist in FB_CtrlModule. Not overrule.
(*
// overrule error always from base -> no EOFF State!! in EOFF go to OFF
IF (me.StateMachine.intStateNext = cSTA_EOFFBusy) THEN
	IF (me.StateMachine.intState=cSTA_OFF) THEN
		me.StateMachine.intStateNext := cSTA_OFF;
	ELSE // stay in OFF
		me.StateMachine.intStateNext := cSTA_OFFBusy;
	END_IF
*)
IF (me.Alarm.eActivAlmClass=E_AlmClass.STOP) AND (me.StateMachine.intStateNext<>cSTA_Error)
		AND ((me.StateMachine.intState = cSTA_RUN) OR (me.StateMachine.intState = cSTA_RUNBusy))THEN
	// alarm evt STOP
	me.StateMachine.intStateNext := cSTA_STOPBusy;	
END_IF
END_METHOD

METHOD checkChildAlmClass : BOOL
//------------------------------------------------------------------------------------------------------
// check child alarm classes
// set me alarm class active if at least one child has an EOFF
IF CheckAllChildAlmClass(E_AlmClass.EOFF) THEN
	CIf.Job.eMe_ActivAlmClass := E_AlmClass.EOFF;
	me.Alarm.bolfp := TRUE;
ELSIF CheckAllChildAlmClass(E_AlmClass.OFF) THEN
	CIf.Job.eMe_ActivAlmClass := E_AlmClass.OFF;
	me.Alarm.bolfp := TRUE;
ELSIF CheckAllChildAlmClass(E_AlmClass.STOP) THEN
	CIf.Job.eMe_ActivAlmClass := E_AlmClass.STOP;
	me.Alarm.bolfp := TRUE;
ELSIF CheckAllChildAlmClass(E_AlmClass.TSTOP) THEN
	CIf.Job.eMe_ActivAlmClass := E_AlmClass.TSTOP;
	me.Alarm.bolfp := TRUE;
ELSE
	IF (me.Alarm.bolfp) THEN
		CIf.Job.eMe_ActivAlmClass := E_AlmClass.NONE; // no reset necessary
		me.Alarm.bolfp := FALSE;
	END_IF
END_IF

//------------------------------------------------------------------------------------------------------
// set alarm class parent of childs
//------------------------------------------------------------------------------------------------------
// set alarm class parent of childs in the case of a parent EOFF or me=OFF or EOFF
IF (CIf.Job.eParent_ActivAlmClass=E_AlmClass.EOFF) THEN
	SetAllChildAlmClass(CIf.Job.eParent_ActivAlmClass);
ELSIF(CIf.Job.eMe_ActivAlmClass=E_AlmClass.EOFF) OR (CIf.Job.eMe_ActivAlmClass=E_AlmClass.OFF) THEN
	SetAllChildAlmClass(CIf.Job.eMe_ActivAlmClass);
ELSE
	// no important alarm for child active
	SetAllChildAlmClass(E_AlmClass.NONE);
END_IF
END_METHOD

METHOD PROTECTED checkValidPointer : BOOL
IF (usiNumOfSeq = usiNumOfValidPointerSeqChild) AND (SIf_Cfg<>0) AND (SIf_Par<>0) AND (SIf_Cur<>0) AND (SIf_In<>0) THEN
	checkValidPointer:= TRUE;
ELSE
	// Invalid child pointer
	checkValidPointer:= FALSE;	
	// SIf.Alm[1].strText := 'Invalid pointer'; 
	pfbAlarmCtrl^.setAlarm(CIf.Info.intCtrlId,1,0,ADR(SIf_MOD.Alm),E_AlmState.RST,CIf.Job.eMe_ActivAlmClass);	
END_IF
END_METHOD

METHOD PROTECTED CtrlInit : BOOL
VAR
	ii: INT;
END_VAR
SUPER^.CtrlInit();

// Initialize all child controller
// Childs are listed in list of sequences
FOR ii:=0 TO usiNumOfSeq-1 BY 1 DO	
	aListOfSeq[ii].pCIF := THIS^.AddChild(aListOfSeq[ii].pChild^);
END_FOR
END_METHOD

METHOD FB_init : BOOL
VAR_INPUT
	///if TRUE, the retain variables are initialized (warm start / cold start)
	bInitRetains: BOOL;
	///if TRUE, the instance afterwards gets moved into the copy code (online change)
	bInCopyCode: BOOL;
END_VAR
VAR
	ii: UINT;
END_VAR
// to manually change in new FUB implementation!!!
// define valid commands for this controller
FOR ii:= 0 TO (SIZEOF(CIf.Job.aCmdList)/SIZEOF(CIf.Job.aCmdList[0])-1) BY 1 DO
	IF (CIf.Job.aCmdList[ii].intCmd=cCMD_INITIALIZED) THEN
		// found first empty array element
		EXIT;
	END_IF
END_FOR

CIf.Job.aCmdList[ii].intCmd := cCMD_RUN;
CIf.Job.aCmdList[ii].strName := 'Run'; 
CIf.Job.aCmdList[ii].bolAvailable := TRUE;
ii := ii +1;
CIf.Job.aCmdList[ii].intCmd := cCMD_STOP;
CIf.Job.aCmdList[ii].strName := 'Stop'; 
CIf.Job.aCmdList[ii].bolAvailable := TRUE;
ii := ii +1;

// set name of class/typ
CIf.Info.strType := 'FB_CtrlModule'; 

// set alarm class
SIf_MOD.Alm[1].eAlmClass := E_AlmClass.STOP;
SIf_MOD.Alm[1].strText := 'Invalid pointer';
SIf_MOD.Alm[2].eAlmClass := E_AlmClass.OFF;
SIf_MOD.Alm[2].strText := 'Communication error to line control'; 
SIf_MOD.Alm[3].eAlmClass := E_AlmClass.EOFF;
SIf_MOD.Alm[3].strText := 'Emergency off active'; 
SIf_MOD.Alm[4].eAlmClass := E_AlmClass.OFF;
SIf_MOD.Alm[4].strText := 'General error active'; 
SIf_MOD.Alm[5].eAlmClass := E_AlmClass.OFF;
SIf_MOD.Alm[5].strText := 'Timeout start group '; 
SIf_MOD.Alm[6].eAlmClass := E_AlmClass.OFF;
SIf_MOD.Alm[6].strText := 'Timeout stop group '; 

//*******************************************************************************
// initial values
//*******************************************************************************
udinTimeToggle_ms := 0;
// software configuration
CIf.SwCfg.bolExist := TRUE;
CIf.SwCfg.bolSimulation := FALSE;

// No initialization for cfg and par in this base module!
// Pointer address of the property is not defined at this time
END_METHOD

METHOD PROTECTED getCmdState : STRING
VAR_INPUT
	intCmdState: INT;
	bolState: BOOL;
END_VAR
getCmdState := SUPER^.getCmdState(intCmdState:=intCmdState,bolState:=bolState); // get global/base defined cmds/states
IF (getCmdState='') THEN // global not defined get local
	// get string cmd/state string information in runtime
	IF (bolState=FALSE) THEN
		// cmd's
	ELSE
	
	// cmd's
		CASE intCmdState OF	
			// SUB States
			cSTA_SUB_INITIALIZED:
				getCmdState := 'cSTA_SUB_INITIALIZED';
			cSTA_SUB_SEND_GROUP_CMD:
				getCmdState := 'cSTA_SUB_SEND_GROUP_CMD';
			cSTA_SUB_CHECK_GROUP_STATUS:
				getCmdState := 'cSTA_SUB_CHECK_GROUP_STATUS';
			cSTA_SUB_WAIT:
				getCmdState := 'cSTA_SUB_WAIT';
			cSTA_SUB_FINISHED:
				getCmdState := 'cSTA_SUB_FINISHED';
		END_CASE;
	END_IF
END_IF
END_METHOD

METHOD PROTECTED IoInBridge : BOOL
// Inputs from global module for general supervision (no physical inputs)
SIf_In^.bolEmergencyOffOk.map := THIS^.In_bolEmergencyOffOk;
SIf_In^.bolNoGeneralError.map := THIS^.In_bolNoGeneralError;

IF (CIf.SwCfg.bolSimulation = FALSE) THEN
	getInBol(CIf.Job.bolIoForce,ADR(SIf_In^.bolEmergencyOffOk));
	getInBol(CIf.Job.bolIoForce,ADR(SIf_In^.bolNoGeneralError));
ELSE
	//simulation of global IO
END_IF
END_METHOD

METHOD PROTECTED IoOutBridge : BOOL
// digitale and analoge inputs read from hardware or forcing
IF (CIf.SwCfg.bolSimulation = FALSE) THEN
	// check interlocks to prevent damages
	IF (CIf.Job.bolIlkOverwrite=FALSE) THEN
	;
	END_IF
END_IF
END_METHOD

PROPERTY SIf_Cfg : POINTER TO T_Ctrl_SIf_MOD_Cfg
GET
SIf_Cfg:= SIf_MOD.Cfg;
END_GET
SET
SIf_MOD.Cfg := SIf_Cfg;
END_SET
END_PROPERTY

PROPERTY SIf_Cur : POINTER TO T_Ctrl_SIf_MOD_Cur
GET
SIf_Cur:= SIf_MOD.Cur;
END_GET
SET
SIf_MOD.Cur := SIf_Cur;
END_SET
END_PROPERTY

PROPERTY SIf_In : POINTER TO T_Ctrl_SIf_MOD_In
GET
SIf_In:= SIf_MOD.In;
END_GET
SET
SIf_MOD.In := SIf_In;
END_SET
END_PROPERTY

PROPERTY SIf_Par : POINTER TO T_Ctrl_SIf_MOD_Par
GET
SIf_Par:= SIf_MOD.Par;
END_GET
SET
SIf_MOD.Par := SIf_Par;
END_SET
END_PROPERTY

METHOD PROTECTED sta_EOFF : BOOL
// state implemetation
//--------------------------------------------------------------------------------------
// Entry action
	IF (me.StateMachine.intState<>me.StateMachine.intStateLastCycle) THEN
		me.StateMachine.intStateLastCycle := me.StateMachine.intState;	
	END_IF

//--------------------------------------------------------------------------------------
// Cyclic action
	IF (me.StateMachine.intState=me.StateMachine.intStateLastCycle) THEN		
		
		// As long as the EMO is not reseted!
		IF NOT (SIf_In^.bolEmergencyOffOk.intern) THEN
			// Clear pending and new commands cyclic to prevent automatic recovery!
			CIf.Job.intACmd := BASE_PLC.cCMD_DONE;
			CIf.Job.intMCmd := BASE_PLC.cCMD_DONE;
		END_IF
	
		// State Change Condition
		IF (SIf_In^.bolEmergencyOffOk.intern) AND (me.Alarm.eActivAlmClass<>E_AlmClass.EOFF) AND (me.intCmd<>BASE_PLC.cCMD_EOFF) AND (me.intCmd<>BASE_PLC.cCMD_DONE) THEN
			me.StateMachine.intStateNext := cSTA_OFF;
		END_IF
	END_IF

//--------------------------------------------------------------------------------------
// Exit action
	IF (me.StateMachine.intState<>me.StateMachine.intStateNext) THEN
		;
	END_IF
END_METHOD

METHOD PROTECTED sta_EOFFBusy : BOOL
// state implemetation
//--------------------------------------------------------------------------------------
// Entry action
	IF (me.StateMachine.intState<>me.StateMachine.intStateLastCycle) THEN
		me.StateMachine.intStateLastCycle := me.StateMachine.intState;
	END_IF

//--------------------------------------------------------------------------------------
// Cyclic action
	IF (me.StateMachine.intState=me.StateMachine.intStateLastCycle) THEN
		
		// In case of an emergency, set all childs to off 
		// Set in cyclic action because of possible errors or manual/auto changes!
		SUPER^.SetAllChildCmd(BASE_PLC.cCMD_OFF);

		// check if all childs have reached the state
		IF CheckAllChildState(cSTA_OFF) THEN
			me.StateMachine.intStateNext := cSTA_EOFF;
		END_IF
	END_IF

//--------------------------------------------------------------------------------------
// Exit action
	IF (me.StateMachine.intState<>me.StateMachine.intStateNext) THEN
		;
	END_IF
END_METHOD

METHOD PROTECTED sta_ERROR : BOOL
// state implemetation
//--------------------------------------------------------------------------------------
// Entry action
	IF (me.StateMachine.intState<>me.StateMachine.intStateLastCycle) THEN
		me.StateMachine.intStateHistory := me.StateMachine.intStateLastCycle; // -> possibillity to go back to state before error
		me.StateMachine.intStateLastCycle := me.StateMachine.intState;
		// Clear pending command to prevent automatic recovery!
		CIf.Job.intACmd:=cSTA_DONE;
		// In case on an error, set all childs to off
		SetAllChildCmd(cCMD_OFF);
	END_IF

//--------------------------------------------------------------------------------------
// Cyclic action
	IF (me.StateMachine.intState=me.StateMachine.intStateLastCycle) THEN
		
		;
		// State Change Condition
		IF ((CIf.Job.bolAlmReset = TRUE) AND (CheckAllChildState(cSTA_OFF))) THEN
			me.StateMachine.intStateNext := cSTA_ERRORQuit;
		END_IF
	END_IF

//--------------------------------------------------------------------------------------
// Exit action
	IF (me.StateMachine.intState<>me.StateMachine.intStateNext) THEN
		;
	END_IF
END_METHOD

METHOD PROTECTED sta_OFF : BOOL
// state implemetation
//--------------------------------------------------------------------------------------
// Entry action
	IF (me.StateMachine.intState<>me.StateMachine.intStateLastCycle) THEN
		me.StateMachine.intStateLastCycle := me.StateMachine.intState;
		;		
	END_IF

//--------------------------------------------------------------------------------------
// Cyclic action
	IF (me.StateMachine.intState=me.StateMachine.intStateLastCycle) THEN
				
		// State Change Condition
		IF (me.Alarm.eActivAlmClass<>E_AlmClass.EOFF) AND (me.Alarm.eActivAlmClass<>E_AlmClass.OFF) THEN
			IF (me.intCmd=cCMD_RUN) THEN 
				me.StateMachine.intStateNext := cSTA_RUNBusy;
			END_IF
		END_IF
	END_IF

//--------------------------------------------------------------------------------------
// Exit action
	IF (me.StateMachine.intState<>me.StateMachine.intStateNext) THEN
		;
	END_IF
END_METHOD

METHOD PROTECTED sta_RUN : BOOL
// state implemetation
//--------------------------------------------------------------------------------------
// Entry action
	IF (me.StateMachine.intState<>me.StateMachine.intStateLastCycle) THEN
		me.StateMachine.intStateLastCycle := me.StateMachine.intState;
		;
	END_IF

//--------------------------------------------------------------------------------------
// Cyclic action
	IF (me.StateMachine.intState=me.StateMachine.intStateLastCycle) THEN

		// Simulation
		IF (CIf.SwCfg.bolSimulation) THEN
			;
		END_IF

		// State Change Condition	
		IF (me.intCmd=cCMD_STOP)  THEN
			me.StateMachine.intStateNext :=  cSTA_STOPBusy;	
		END_IF

	END_IF

//--------------------------------------------------------------------------------------
// Exit action
	IF (me.StateMachine.intState<>me.StateMachine.intStateNext) THEN
		;
	END_IF
END_METHOD

METHOD PROTECTED sta_RUNBusy : BOOL
VAR
	ii: INT;
	bolFurtherGrpExist: BOOL;
END_VAR
// state implemetation
//--------------------------------------------------------------------------------------
// Entry action
	IF (me.StateMachine.intState<>me.StateMachine.intStateLastCycle) THEN
		me.StateMachine.intStateLastCycle := me.StateMachine.intState;
		// Init sub state machine
		me.SubStateMachine.intState := cSTA_SUB_INITIALIZED; 
		me.SubStateMachine.intStateNext := cSTA_SUB_INITIALIZED;
	END_IF

//--------------------------------------------------------------------------------------
// Cyclic action
	IF (me.StateMachine.intState=me.StateMachine.intStateLastCycle) THEN

		// Simulation
		IF (CIf.SwCfg.bolSimulation) THEN
			;
		END_IF
	
		// Start Cycle with substates	
		//--------------------------------------------------------------------------------------
		// sub state machine for sequence
		CASE me.SubStateMachine.intState OF
			//--------------------------------------------------------------------------------------
			cSTA_SUB_INITIALIZED:
			
				// Loop over all registered childs
				FOR ii:=0 TO usiNumOfSeq-1 BY 1 DO
					// Clear checked flag		
					aListOfSeq[ii].bolChecked:= FALSE;
				END_FOR
				uinGroupIndex:= 1;
				me.SubStateMachine.intStateNext := cSTA_SUB_SEND_GROUP_CMD;
				
			cSTA_SUB_SEND_GROUP_CMD:
				
				intCheckCounter:= 0;
				// Loop over all registered childs
				FOR ii:=0 TO usiNumOfSeq-1 BY 1 DO
					// If child is associated for the current group index		
					IF (aListOfSeq[ii].uinGroupRun = uinGroupIndex) THEN
						// Send defined command
						aListOfSeq[ii].pCIF^.Job.intACmd:= aListOfSeq[ii].intCmdSeqRun;
						intCheckCounter:= intCheckCounter + 1;
					END_IF			
				END_FOR
				// Change state
				me.SubStateMachine.intStateNext := cSTA_SUB_CHECK_GROUP_STATUS;
			
			
			cSTA_SUB_CHECK_GROUP_STATUS:
	
				// Loop over all registered childs
				FOR ii:=0 TO usiNumOfSeq-1 BY 1 DO
					// If child is associated for the current group index		
					IF (aListOfSeq[ii].uinGroupRun = uinGroupIndex) THEN
						// Check defined status and if child not already checked
						IF (((aListOfSeq[ii].pCIF^.Job.intState = aListOfSeq[ii].intStatusSeqRun) OR 
						(aListOfSeq[ii].pCIF^.Job.intState = aListOfSeq[ii].intStatusSeqRun2)) AND (aListOfSeq[ii].bolChecked = FALSE)) THEN
							aListOfSeq[ii].bolChecked:= TRUE;
							intCheckCounter:= intCheckCounter - 1;
						END_IF				
					END_IF			
				END_FOR
				
				// All childs in group has the right state
				IF (intCheckCounter <= 0) THEN		
					bolFurtherGrpExist:= FALSE;
					// Check if a further group exist!	
					FOR ii:=0 TO usiNumOfSeq-1 BY 1 DO	
						IF (aListOfSeq[ii].uinGroupRun > uinGroupIndex) THEN
							bolFurtherGrpExist:= TRUE;
							EXIT;
						END_IF			
					END_FOR
					// further group exist
					IF (bolFurtherGrpExist = TRUE) THEN
						IF (uinGroupIndex < uinMaxNrOfGroups) THEN			
							me.SubStateMachine.intStateNext := cSTA_SUB_WAIT;	
						END_IF
					ELSE
						me.SubStateMachine.intStateNext := cSTA_SUB_FINISHED;		
					END_IF
				END_IF

			cSTA_SUB_WAIT:
				
				IF (me.SubStateMachine.udiTimeInState_ms >= SIf_Par^.aListOfRunGrpWaitTime_ms[uinGroupIndex-1]) THEN
					// Inc. group index 
					uinGroupIndex:= uinGroupIndex + 1;	
					// Change state, send command for next group
					me.SubStateMachine.intStateNext := cSTA_SUB_SEND_GROUP_CMD;
				END_IF
			
			cSTA_SUB_FINISHED:
					;		
		END_CASE
		
		// Check time out error
		IF (me.SubStateMachine.udiTimeInState_ms > (SIf_Par^.aListOfRunGrpWaitTime_ms[uinGroupIndex-1] + 30000)) THEN
			// SIf_MOD.Alm[5].strText := 'Timeout start group '; 
			pfbAlarmCtrl^.setAlarm(CIf.Info.intCtrlId,5,uinGroupIndex,ADR(SIf_MOD.Alm),E_AlmState.RST,CIf.Job.eMe_ActivAlmClass);
		END_IF
		
		// State Change Condition
		IF (me.SubStateMachine.intState = cSTA_SUB_FINISHED) THEN
			me.StateMachine.intStateNext := cSTA_RUN;
		ELSIF (me.intCmd=cCMD_STOP) THEN
			me.StateMachine.intStateNext :=  cSTA_STOPBusy;	
		END_IF
	END_IF

//--------------------------------------------------------------------------------------
// Exit action
	IF (me.StateMachine.intState<>me.StateMachine.intStateNext) THEN
		;
	END_IF
END_METHOD

METHOD PROTECTED sta_STOP : BOOL
// state implemetation
//--------------------------------------------------------------------------------------
// Entry action
	IF (me.StateMachine.intState<>me.StateMachine.intStateLastCycle) THEN
		me.StateMachine.intStateLastCycle := me.StateMachine.intState;
		
	END_IF


//--------------------------------------------------------------------------------------
// Cyclic action
	IF (me.StateMachine.intState=me.StateMachine.intStateLastCycle) THEN
		
		;	
		// State Change Condition
		IF (me.Alarm.eActivAlmClass<>E_AlmClass.STOP) THEN
			IF (me.intCmd=cCMD_RUN) THEN
				me.StateMachine.intStateNext :=  cSTA_RUNBusy;
			END_IF
		END_IF
	END_IF

//--------------------------------------------------------------------------------------
// Exit action
	IF (me.StateMachine.intState<>me.StateMachine.intStateNext) THEN
		;
	END_IF
END_METHOD

